	IF (MANUAL_SELECTED AND OP10B_M_PICK_PART_OK) OR OP10B_A_PICK_PART_OK THEN
		OP10B_PICK_PART_OK								:= TRUE;
		OP10B_A_ORING_INSERTION_DONE					:= TRUE;
		OP10B_Gripper_Rotate_Complete					:= TRUE;
		OP10B_Camera_Zone_Safe							:= TRUE;(*(OP10A_SRV_RH_BDYANG_CMR_FB OR OP10A_BDY2_PCK_BYPAS) AND 
															(OP10A_SRV_LH_BDYANG_CMR_FB OR OP10A_BDY1_PCK_BYPAS);*)
	ELSE
		OP10B_PICK_PART_OK								:= FALSE;
		OP10B_Gripper_Rotate_Complete					:= FALSE;
		OP10B_Camera_Zone_Safe							:= FALSE;
		OP10B_A_ORING_INSERTION_DONE					:= FALSE;		
	END_IF

	IF (MANUAL_SELECTED AND OP10B_M_PICK_PART_NOK) OR OP10B_A_PICK_PART_NOK THEN
		OP10B_PICK_PART_NOK								:= TRUE;
	ELSE
		OP10B_PICK_PART_NOK								:= FALSE;		
	END_IF

	IF (MANUAL_SELECTED AND OP10B_M_CAMERA_OK) OR OP10B_A_CAMERA_OK THEN
		OP10B_READY_TO_INSERT_ORING						:= TRUE;
		OP10B_Place_Zone_Safe							:= (OP10B_SRV_LH_BDYANG_WRK_FB OR OP10B_BDY1_PCK_BYPAS) AND 
															(OP10B_SRV_RH_BDYANG_WRK_FB OR OP10B_BDY2_PCK_BYPAS);
		OP10B_ROTATION_COMPLETE							:= TRUE;
		OP10B_O_Ring_Zone_Safe							:=  (OP10B_SRV_LH_BDYANG_FITRE_FB OR OP10B_BDY1_PCK_BYPAS) AND 
															(OP10B_SRV_RH_BDYANG_FITRE_FB OR OP10B_BDY2_PCK_BYPAS) AND 
																OP10B_CYL_RDY_TO_PLC;

		IF OP10B_ROBO_CNTRL.BDY_MVE_PLC_POS THEN
		OP10B_A_PLACE_IN_CONVEYOR						:= TRUE;			
		END_IF
		
		IF OP10B_Camera_Trigger THEN
		OP10B_CAMERA_OK									:= TRUE;	
		END_IF											
															
	ELSE                                            	
		OP10B_CAMERA_OK									:= FALSE;
		OP10B_READY_TO_INSERT_ORING						:= FALSE;
		OP10B_O_Ring_Zone_Safe							:= FALSE;
		OP10B_Place_Zone_Safe							:= FALSE;
		OP10B_A_PLACE_IN_CONVEYOR						:= FALSE;
		OP10B_ROTATION_COMPLETE							:= FALSE;		
	END_IF

	IF (MANUAL_SELECTED AND OP10B_M_CAMERA_NOK) OR OP10B_A_CAMERA_NOK AND OP10B_Camera_Trigger THEN
		OP10B_CAMERA_NOK								:= TRUE;
	ELSE
		OP10B_CAMERA_NOK								:= FALSE;		
	END_IF	 

 	IF (MANUAL_SELECTED AND OP10B_M_ORING_INSERTION_DONE) OR OP10B_A_ORING_INSERTION_DONE THEN
		OP10B_ORING_INSERTION_DONE						:= TRUE;
	ELSE
		OP10B_ORING_INSERTION_DONE						:= FALSE;		
	END_IF 
   
  	IF (MANUAL_SELECTED AND OP10B_M_PLACE_IN_CONVEYOR) OR OP10B_A_PLACE_IN_CONVEYOR THEN
		OP10B_PLACE_IN_CONVEYOR							:= TRUE;
	ELSE
		OP10B_PLACE_IN_CONVEYOR							:= FALSE;		
	END_IF

	OP10B_GRIPPER_OPEN									:= (OP10B_A_SRV_LH_GRPHME_FB OR OP10B_BDY1_PCK_BYPAS )AND (OP10B_A_SRV_RH_GRPHME_FB OR OP10B_BDY2_PCK_BYPAS) AND NOT OP10B_ROBO_Gripper_Close;
	OP10B_GRIPPER_CLOSE									:= (OP10B_A_SRV_LH_GRPWRK_FB OR  OP10B_BDY1_PCK_BYPAS)AND (OP10B_A_SRV_RH_GRPWRK_FB OR OP10B_BDY2_PCK_BYPAS) AND OP10B_ROBO_Gripper_Close;

	OP10B_Reject_Zone_Safe								:= 1;//NOT OP10A_Rbt_In_Reject_Zone;
	
//############################		OP10B STATION ENABLE CONDITION		##########################

	OP10B_STN_MOVER					:= MOVER_POSITION[OP10B_XTS_POS_NO];

	IF AUTO_WITH_XTS THEN
	IF 	OP10B_STN_MOVER>0 THEN
	IF NOT END_OF_CYCLE THEN		
	OP10B_STN_ENABLE				:= MOVER_POS_RECHED[OP10B_STN_MOVER] AND ((MOVER_CMP_STATUS[OP10B_STN_MOVER][1]=0)OR 
										(MOVER_CMP_STATUS[OP10B_STN_MOVER][2]=0))AND STATION_ENABLE_CONTROL AND NOT 
											(I10B_BDY1_PRSN_MOVER_I1001_5 OR I10B_BDY2_PRSN_MOVER_I1001_6);
  	
  
ELSE
	MOVER_CMP_STATUS[OP10B_STN_MOVER][1]					:=5;
	MOVER_CMP_STATUS[OP10B_STN_MOVER][2]					:=5;
	STATION_DONE[OP10B_STN_MOVER][OP10B_XTS_POS_NO]			:= TRUE;	
	END_IF
	ELSE	
	OP10B_STN_ENABLE				:= FALSE;
	END_IF
	END_IF

END_PROGRAM

// ---- POUs/Programs/OP10A_Bowl/Bowl_Control.TcPOU
PROGRAM Bowl_Control
VAR
	OP10A_Bowl: ModbusRtuMasterV2_KL6x22B;
	Write_Reg: UINT;
	Read: UINT;
	W_Trig	: BOOL;
	Read_Reg : UINT;
	R_Trig	: BOOL;
	Rsad:BOOL;
	Trigger: BOOL;
	R_Edge	: R_TRIG;
	reg: WORD;
	writereg: WORD;
END_VAR

//R_Edge(CLK:=W_Trig);

OP10A_Bowl.WriteSingleRegister(
	UnitID:= 1, 
	Quantity:=1 , 
	MBAddr:= writereg, 
	cbLength:= SIZEOF(Write_Reg), 
	pMemoryAddr:= ADR(Write_Reg), 
	AuxQuantity:= , 
	AuxMBAddr:= , 
	AuxcbLength:= , 
	pAuxMemoryAddr:= , 
	Execute:=W_Trig,//R_Edge.Q , 
	Timeout:= , 
	BUSY=> , 
	Error=> , 
	ErrorId=> , 
	cbRead=> );


OP10A_Bowl.ReadInputRegs(
	UnitID:= 1, 
	Quantity:=1 , 
	MBAddr:= reg, 
	cbLength:= SIZEOF(Read), 
	pMemoryAddr:= ADR(Read), 
	AuxQuantity:= , 
	AuxMBAddr:= , 
	AuxcbLength:= , 
	pAuxMemoryAddr:= , 
	Execute:=Rsad,//R_Edge.Q , 
	Timeout:= , 
	BUSY=> , 
	Error=> , 
	ErrorId=> , 
	cbRead=> );
		
	
OP10A_Bowl.ReadInputRegs(
	UnitID:= 1, 
	Quantity:=1 , 
	MBAddr:= 16#01, 
	cbLength:= SIZEOF(Read_Reg), 
	pMemoryAddr:= ADR(Read_Reg), 
	AuxQuantity:= , 
	AuxMBAddr:= , 
	AuxcbLength:= , 
	pAuxMemoryAddr:= , 
	Execute:= R_Trig, 
	Timeout:= , 
	BUSY=> , 
	Error=> , 
	ErrorId=> , 
	cbRead=> );

END_PROGRAM

// ---- POUs/Programs/OP10/OP10A_Camera_FB.TcPOU
PROGRAM OP10A_Camera_FB
VAR
	OP10A_LH_Camera 			        : FB_Cognex_ProfiNET_1;
	
	OP10A_LH_Acquisition_Status AT %I*    :Acquisition_Status;
	OP10A_LH_Inspection_Status  AT %I*    :Inspection_Status;	
	OP10A_LH_Acquisition_ID     AT %I*    :UINT;
	OP10A_LH_Inspection_ID   	 AT %I*  :UINT;
	OP10A_LH_Error_code      	 AT %I*  :UINT;
	OP10A_LH_Current_Job_ID  	 AT %I*  :UINT;
	OP10A_LH_Result_code     	 AT %I*  :UINT;
	OP10A_LH_Cam_Result      	 AT %I*  :ARRAY[0..63] OF BYTE;	
	OP10A_LH_Acquisition_Control AT %Q*  : Acquisition_Control;
	OP10A_LH_Inspection_Control  AT %Q*  : Inspection_Control;
	OP10A_LH_Command_word		AT %Q*  : UINT;
	OP10A_LH_Union                       : UNION_64Byte;

	OP10A_RH_Camera 			          : FB_Cognex_ProfiNET_1;

	
	OP10A_RH_Acquisition_Status AT %I*    :Acquisition_Status;
	OP10A_RH_Inspection_Status  AT %I*    :Inspection_Status;	
	OP10A_RH_Acquisition_ID     AT %I*    :UINT;
	OP10A_RH_Inspection_ID   	 AT %I*  :UINT;
	OP10A_RH_Error_code      	 AT %I*  :UINT;
	OP10A_RH_Current_Job_ID  	 AT %I*  :UINT;
	OP10A_RH_Result_code     	 AT %I*  :UINT;
	OP10A_RH_Cam_Result      	 AT %I*  :ARRAY[0..63] OF BYTE;	
	OP10A_RH_Acquisition_Control AT %Q*  : Acquisition_Control;
	OP10A_RH_Inspection_Control  AT %Q*  : Inspection_Control;
	OP10A_RH_Command_word		AT %Q*  : UINT;
	OP10A_RH_Union                       : UNION_64Byte;
	
	OP10_A_Empty_Camera_1	      : FB_Cognex_ProfiNET_1;
	
	
	OP10A_Empty_Cam_1_Acquisition_Status   AT %I*  :Acquisition_Status;
	OP10A_Empty_Cam_1_Inspection_Status    AT %I*  :Inspection_Status;	
	OP10A_Empty_Cam_1_Acquisition_ID       AT %I*  :UINT;
	OP10A_Empty_Cam_1_Inspection_ID   	 AT %I*  :UINT;
	OP10A_Empty_Cam_1_Error_code      	 AT %I*  :UINT;
	OP10A_Empty_Cam_1_Current_Job_ID  	 AT %I*  :UINT;
	OP10A_Empty_Cam_1_Result_code     	 AT %I*  :UINT;
	OP10A_Empty_Cam_1_Result      	 AT %I*  :ARRAY[0..63] OF BYTE;
	
	OP10A_Empty_Cam_1_Acquisition_Control AT %Q*  : Acquisition_Control;
	OP10A_Empty_Cam_1_Inspection_Control  AT %Q*  : Inspection_Control;
	OP10A_Empty_Cam_1_Command_word		AT %Q*  : UINT;
	Error_status_Cam_1						      : STRING;
	OP10A_Empty_Cam_1_Target_Job_ID				  : UINT;
	OP10A_Empty_Cam_1_Loaded_Job_ID		    	  : UINT;
	OP10A_Empty_Cam_1_Union                       : UNION_64Byte;
	OP10A_Empty_Cam_1_Job_Change_Complete		  : BOOL;
	OP10A_Empty_Cam_1_Job_Change_Error   		  : BOOL;
	OP10A_Empty_Cam_1_Picture_Taken      		  : BOOL;	
	
END_VAR

OP10A_LH_Camera (
	tTimeout:= , 
	sJob_Name:= , 
	camera_ready=> OP10A_LH_Camera_Ready,
	Camera_online=> OP10A_LH_Camera_Online,
	stCognex_record_status:=OP10A_LH_Acquisition_Status, 
	Acquisition_ID:=OP10A_LH_Acquisition_ID , 
	stCognex_Inspection_status:=OP10A_LH_Inspection_Status, 
	Error_Code:=OP10A_LH_Error_code , 
	wcommand_control_in:= OP10A_LH_Current_Job_ID, 
	aResults_64_Bytes:= OP10A_LH_Cam_Result, 
	number_of_inspections:=OP10A_LH_Inspection_ID , 
	iresult_code:= OP10A_LH_Result_code, 
	bTarget_job_ID:=OP10A_LH_Target_Job_ID , 
	Error_Status_message=> OP10A_LH_Error_status, 
	bError=> OP10A_LH_Camera_Error, 
	stCognex_record_control=>OP10A_LH_Acquisition_Control , 
	stCognex_inspection_control=>OP10A_LH_Inspection_Control , 
	wCommandControl_out=>OP10A_LH_Command_word , 
	aUser_data_64_Byte=> OP10A_LH_Union.aArrayOfByte, 
	bJob_loading_completed=>OP10A_LH_Job_Change_Complete , 
	bJob_load_failed=>OP10A_LH_Job_Change_Error , 
	bInspection_Result_IO=>  , 
	bInspection_Result_NIO=> , 
	bTXTSM_Error_Job_Change=> OP10A_LH_Job_Change_Error, 
	bPictureTakenComplete=> OP10A_LH_Picture_Taken, 
	Loaded_Job_ID=>OP10A_LH_Loaded_Job_ID	 , 
	bClear_Error:= HMI_Reset, 
	bJob_change_start:= OP10A_LH_Camera_Job_Change_start, 
	TXTSM_camera_not_online=>OP10A_LH_Camera_Error	 , 
	bTrigger_start:= OP10A_LH_Camera_Trigger );
	
OP10A_RH_Camera (
	tTimeout:= , 
	sJob_Name:= , 
	camera_ready=> OP10A_RH_Camera_Ready,
	Camera_online=> OP10A_RH_Camera_Online,
	stCognex_record_status:=OP10A_RH_Acquisition_Status, 
	Acquisition_ID:=OP10A_RH_Acquisition_ID , 
	stCognex_Inspection_status:=OP10A_RH_Inspection_Status, 
	Error_Code:=OP10A_RH_Error_code , 
	wcommand_control_in:= OP10A_RH_Current_Job_ID, 
	aResults_64_Bytes:= OP10A_RH_Cam_Result, 
	number_of_inspections:=OP10A_RH_Inspection_ID , 
	iresult_code:= OP10A_RH_Result_code, 
	bTarget_job_ID:=OP10A_RH_Target_Job_ID , 
	Error_Status_message=> OP10A_RH_Error_status, 
	bError=> OP10A_RH_Camera_Error, 
	stCognex_record_control=>OP10A_RH_Acquisition_Control , 
	stCognex_inspection_control=>OP10A_RH_Inspection_Control , 
	wCommandControl_out=>OP10A_RH_Command_word , 
	aUser_data_64_Byte=> OP10A_RH_Union.aArrayOfByte, 
	bJob_loading_completed=>OP10A_RH_Job_Change_Complete , 
	bJob_load_failed=>OP10A_RH_Job_Change_Error , 
	bInspection_Result_IO=>  , 
	bInspection_Result_NIO=> , 
	bTXTSM_Error_Job_Change=> OP10A_RH_Job_Change_Error, 
	bPictureTakenComplete=> OP10A_RH_Picture_Taken, 
	Loaded_Job_ID=>OP10A_RH_Loaded_Job_ID	 , 
	bClear_Error:= HMI_Reset, 
	bJob_change_start:= OP10A_RH_Camera_Job_Change_start, 
	TXTSM_camera_not_online=>OP10A_RH_Camera_Error	 , 
	bTrigger_start:= OP10A_RH_Camera_Trigger );	
	
OP10_A_Empty_Camera_1(
	tTimeout:= , 
	sJob_Name:= , 
	camera_ready=> OP10A_Empty_Cam_1_Camera_Ready,
	Camera_online=> OP10A_Empty_Cam_1_Camera_Online,
	stCognex_record_status:=OP10A_Empty_Cam_1_Acquisition_Status, 
	Acquisition_ID:=OP10A_Empty_Cam_1_Acquisition_ID , 
	stCognex_Inspection_status:=OP10A_Empty_Cam_1_Inspection_Status, 
	Error_Code:=OP10A_Empty_Cam_1_Error_code , 
	wcommand_control_in:= OP10A_Empty_Cam_1_Current_Job_ID, 
	aResults_64_Bytes:= OP10A_Empty_Cam_1_Result, 
	number_of_inspections:=OP10A_Empty_Cam_1_Inspection_ID , 
	iresult_code:= OP10A_Empty_Cam_1_Result_code, 
	bTarget_job_ID:=OP10A_Empty_Cam_1_Target_Job_ID , 
	Error_Status_message=> Error_status_Cam_1, 
	bError=> OP10A_Empty_Cam_1_Camera_Error, 
	stCognex_record_control=>OP10A_Empty_Cam_1_Acquisition_Control , 
	stCognex_inspection_control=>OP10A_Empty_Cam_1_Inspection_Control , 
	wCommandControl_out=>OP10A_Empty_Cam_1_Command_word , 
	aUser_data_64_Byte=> OP10A_Empty_Cam_1_Union.aArrayOfByte, 
	bJob_loading_completed=>OP10A_Empty_Cam_1_Job_Change_Complete, 
	bJob_load_failed=>OP10A_Empty_Cam_1_Job_Change_Error , 
	bInspection_Result_IO=>  , 
	bInspection_Result_NIO=> , 
	bTXTSM_Error_Job_Change=> OP10A_Empty_Cam_1_Job_Change_Error, 
	bPictureTakenComplete=> OP10A_Empty_Cam_1_Picture_Taken, 
	Loaded_Job_ID=>OP10A_Empty_Cam_1_Loaded_Job_ID	 , 
	bClear_Error:= HMI_Reset, 
	bJob_change_start:= OP10A_Empty_Cam_1_Camera_Job_Change_start, 
	TXTSM_camera_not_online=>OP10A_Empty_Cam_1_Camera_Error	 , 
	bTrigger_start:= OP10A_Empty_Cam_1_Camera_Trigger );

END_PROGRAM

// ---- FB/Cognex_Camera/FB_Cognex_ProfiNET_1.TcPOU
FUNCTION_BLOCK FB_Cognex_ProfiNET_1
VAR_INPUT
	tTimeout						: TIME := T#10S;
	sJob_Name 						: STRING(63) := '';
	stCognex_record_status     		: Acquisition_status;
	Acquisition_ID					: UINT ;//number of shots
	stCognex_Inspection_status 		: Inspection_status;
	Error_Code						: UINT ;
	wcommand_control_in 			: UINT;
    aResults_64_Bytes	     		: ARRAY[0..63] OF BYTE;
    number_of_inspections			: UINT;
	iresult_code					: UINT;
	bClear_Error					: BOOL;	
	bTarget_job_ID					: UINT;
END_VAR

VAR_OUTPUT
	Error_Status_message			:STRING;
	bError							: BOOL := 0;
	stCognex_record_control 		: Acquisition_Control;
	stCognex_inspection_control 	: Inspection_control;
    wCommandControl_out 			: UINT;
    aUser_data_64_Byte 			    : ARRAY[0..63] OF BYTE;
	bJob_loading_completed 		    : BOOL := 0; //FP
	bJob_load_failed        		: BOOL := 0; //FP
	bInspection_Result_IO 			: BOOL := 0; //FP
	bInspection_Result_NIO 			: BOOL := 0; //FP
	bTXTSM_Error_Job_Change 		: BOOL;
	bPictureTakenComplete			: BOOL;
	Loaded_Job_ID					: UINT;
	camera_ready					: BOOL;
	Camera_online					: BOOL;
	TXTSM_camera_not_online 		: BOOL := 0;
END_VAR

VAR_IN_OUT
	bJob_change_start				: BOOL := 0;	
	bTrigger_start					: BOOL := 0;
END_VAR

VAR
	ttimeout_step					: TON;
	tTimeoutStepTrigger			    : TON;
	Resul_ACk_Timer					: TON;
	//JobChange
	job_Change_OK					: R_TRIG;
	job_Change_NOK					: R_TRIG;	
	iStep_Jobchange 				: INT := 0;
	bJob_change_io 					: BOOL:= 0;
	bJob_change_nio 				: BOOL:= 0;
	//Trigger
	Trig_Start						: R_TRIG;
    iStep_Trigger				    : INT := 0;
	bInspection_io 					: BOOL:= 0;
	bInspection_nio 				: BOOL:= 0;
	bHMFPInspection_Completed		: BOOL;//HM_FP_Inspection_Completed
	bHMFNInspection_Completed		: BOOL;//HM_FN_Inspection_Completed
    
    Previous_job_id                 : UINT;   //Job ID for the last job loaded.
    Previous_job_name               : STRING; // Job name of the last job loaded.
END_VAR
VAR_TEMP
	tempaUserData_64_Byte		    : UNION_64Byte;
	bT_in 							: BOOL := FALSE;
	bT_inTrigger					: BOOL := FALSE;
	FPInspection_Completed			: BOOL := FALSE;
	FNInspection_Completed			: BOOL := FALSE;
END_VAR

stCognex_inspection_control.Buffer_Results_Enable 	:= FALSE;
stCognex_inspection_control.Inspection_Results_Ack 	:= FALSE;

Resul_ACk_Timer(IN:=stCognex_inspection_control.Inspection_Results_Ack,PT:=T#100MS);
IF Resul_ACk_Timer.Q THEN
	stCognex_inspection_control.Inspection_Results_Ack:=FALSE;
END_IF

// picture taken complete
bPictureTakenComplete:=stCognex_record_status .Exposure_Complete AND (iStep_Trigger <> 0);
stCognex_record_control.Clear_Exposure_Complete:= stCognex_record_status .Exposure_Complete;

//#########################################################################
//ErrorReset###############################################################
//#########################################################################

bError := stCognex_Inspection_status .Error;
IF bError THEN
	Previous_job_id   := 0;
    Previous_job_name := '';
END_IF

IF stCognex_Inspection_status .Error AND bClear_Error THEN
	stCognex_inspection_control.Clear_Error := TRUE;
ELSE	
	stCognex_inspection_control.Clear_Error := FALSE;
END_IF;

IF NOT stCognex_Inspection_status .Error THEN
	bClear_Error:=FALSE;
END_IF

//#########################################################################
//JobChange################################################################
//#########################################################################

CASE iStep_Jobchange OF 
	0:	//Waiting for bJob_change_start
		bJob_loading_completed := FALSE;
		bJob_load_failed := FALSE;
		bJob_change_io  := FALSE;
		bJob_change_nio := FALSE;

        // Job is still the same.
        IF (TRUE
            AND bJob_change_start
            AND (iStep_Trigger = 0)
            AND (Previous_job_id = bTarget_job_ID )
            AND (Previous_job_name = sJob_Name)
           )
        THEN
			bJob_change_start := FALSE;
            
        // Neuen Job laden.
		ELSIF bJob_change_start AND (iStep_Trigger = 0)THEN
			bJob_change_start := FALSE;
			iStep_Jobchange := 1;
		END_IF;
		
	1://Set Offline
		stCognex_record_control.Set_Offline := TRUE;
		bT_in := TRUE;
		
		IF stCognex_record_status .Online = FALSE 
			AND ( stCognex_record_status .Offline_Bit0 
					OR stCognex_record_status .Offline_Bit1 
					OR stCognex_record_status .Offline_Bit2) 
			THEN
				bT_in := FALSE;
				iStep_Jobchange := 2;
		ELSIF ttimeout_step.Q THEN //Timeout 
				bT_in := FALSE;
				iStep_Jobchange := 8;
		END_IF;
		ttimeout_step(IN:= bT_in, PT:= tTimeout, Q=> , ET=> );
		
	2://Load command(Job ID)
		wCommandControl_out := bTarget_job_ID;//4000;//
		iStep_Jobchange := 3;
		
	3://Set Job name to user data
		//FOR i:=0 TO 63 DO//initalize with 0
		//	aBenutzerdaten_64_Byte[i] := 0;
		//END_FOR;
		tempaUserData_64_Byte.sString := sJob_Name;
		aUser_data_64_Byte := tempaUserData_64_Byte.aArrayOfByte;
		iStep_Jobchange := 4;

	4://Set the Execute Command BIT in the Inspection Control Module.;
		stCognex_inspection_control.Execute_Command := TRUE;
		bT_in := TRUE;
	
		IF stCognex_Inspection_status .Command_Complete AND NOT stCognex_Inspection_status .Command_Executing THEN//Wait for result
			IF stCognex_Inspection_status .Command_Failed THEN//Job load failed 
				bT_in := FALSE;
				iStep_Jobchange := 6;
			ELSE//Job load ok
				bT_in := FALSE;
			iStep_Jobchange := 5;
			END_IF;
		ELSIF ttimeout_step.Q THEN //Timeout 
			bT_in := FALSE;
			iStep_Jobchange := 8;
		END_IF;
		ttimeout_step (IN:= bT_in, PT:= tTimeout, Q=> , ET=> );
		
	5: //Job load ok
			bT_in:= TRUE;
			stCognex_inspection_control.Execute_Command := FALSE;
			bJob_change_io := TRUE;
			bJob_change_nio := FALSE;
            
            Previous_job_id   := wcommand_control_in;
            Previous_job_name := sJob_Name;
			
		IF NOT stCognex_Inspection_status .Command_Executing THEN
			bT_in:= FALSE;
			iStep_Jobchange := 7;
		ELSIF ttimeout_step.Q THEN //Timeout 
			bT_in := FALSE;
			iStep_Jobchange := 8;
		END_IF;
		ttimeout_step(IN:= bT_in, PT:= tTimeout, Q=> , ET=> );
			
	6:	//Job load failed
			bT_in:= TRUE;
			stCognex_inspection_control.Execute_Command := FALSE;
			bJob_change_io := FALSE;
			bJob_change_nio := TRUE;
            
            Previous_job_id   := 0;
            Previous_job_name := '';
			
		IF NOT stCognex_Inspection_status .Command_Executing THEN
			bT_in:= FALSE;
			iStep_Jobchange := 7;
		ELSIF ttimeout_step.Q THEN //Timeout 
			bT_in := FALSE;
			iStep_Jobchange := 8;
		END_IF;
		ttimeout_step(IN:= bT_in, PT:= tTimeout, Q=> , ET=> );
			
	7://Set online 
		bT_in := TRUE;
		stCognex_record_control.Set_Offline := FALSE;
		
		IF stCognex_record_status .Online = TRUE THEN
			iStep_Jobchange := 9;
			bT_in := FALSE;
		ELSIF ttimeout_step.Q THEN //Timeout 
			iStep_Jobchange := 8;
			bT_in := FALSE;
		END_IF;
		ttimeout_step(IN:= bT_in, PT:= tTimeout, Q=> , ET=> );
		
	8://Global Timeout
			stCognex_record_control.Set_Offline := FALSE;
			stCognex_inspection_control.Execute_Command := FALSE;
			bJob_change_io := FALSE;
			bJob_change_nio := TRUE;
			iStep_Jobchange := 9;
			
	9://Set Output signals
	 IF bTarget_job_ID=Loaded_Job_ID  THEN
		bJob_loading_completed:=1;
	 ELSE
	 	bJob_load_failed:=1;
	 END_IF

		//bJob_loading_completed := bJob_change_io;
		//bJob_load_failed := bJob_change_nio;
		iStep_Jobchange := 0;
	ELSE //CASE JobChange default
		
	iStep_Jobchange := 0;
	
END_CASE;

//output error messages Job-change

IF bJob_change_nio THEN
	bTXTSM_Error_Job_Change := TRUE;
	Previous_job_id   := 0;
    Previous_job_name := '';
ELSIF (bJob_change_io AND NOT bJob_change_nio) OR bClear_Error THEN
	bTXTSM_Error_Job_Change := FALSE;
END_IF;

	// IF bTarget_job_ID=Loaded_Job_ID  THEN
	//	bJob_loading_completed:=1;
	// ELSE
	// 	bJob_load_failed:=1;
	// END_IF
//#########################################################################
//Trigger##################################################################
//#########################################################################
//Inspection_Completed edge (Toggle)
FPInspection_Completed 		:= stCognex_Inspection_status .Inspection_Completed AND NOT bHMFPInspection_Completed ;
bHMFPInspection_Completed 	:= stCognex_Inspection_status .Inspection_Completed;

FNInspection_Completed := NOT stCognex_Inspection_status .Inspection_Completed AND bHMFNInspection_Completed ;
bHMFNInspection_Completed := 	stCognex_Inspection_status .Inspection_Completed;
//Camera waiting for result:
IF iStep_Trigger = 2
	 OR iStep_Trigger = 3
	 OR iStep_Trigger = 4 
THEN
	IF (FPInspection_Completed OR FNInspection_Completed) THEN
        IF stCognex_Inspection_status .Results_Valid THEN // stCognex_Inspection_status .Job_Pass THEN
		    bInspection_io  := TRUE;
		    bInspection_nio := FALSE;
			stCognex_inspection_control.Inspection_Results_Ack :=TRUE;
        ELSE
		    bInspection_io  := FALSE;
		    bInspection_nio := TRUE;
			stCognex_inspection_control.Inspection_Results_Ack :=TRUE;
        END_IF
	END_IF
(* PHU: von ARU
	IF (FPInspection_Completed OR FNInspection_Completed) AND stCognex_Inspektionsstatus.Job_Pass THEN
		bInspection_io := TRUE; 
	ELSIF (FPInspection_Completed OR FNInspection_Completed) AND NOT stCognex_Inspektionsstatus.Job_Pass THEN
		bInspection_nio := TRUE; 
	END_IF
*)
END_IF
CASE iStep_Trigger OF 
	0:	//Waiting for bTrigger_start
		bInspection_Result_IO := FALSE;
		bInspection_Result_NIO := FALSE;
		bInspection_io  := FALSE;
		bInspection_nio := FALSE;
		
		Trig_Start(CLK:=bTrigger_start);
		IF Trig_Start.Q AND (iStep_Jobchange = 0) AND NOT bTXTSM_Error_Job_Change THEN
			bTrigger_start := FALSE;
			iStep_Trigger := 1;
		END_IF;
	1://Enable External Trigger
		stCognex_record_control.Trigger_Enable := TRUE;
		stCognex_record_control.Trigger := FALSE;
		//stCognex_Aufnahmesteuerung.Trigger := FALSE;
		
		IF  stCognex_record_status .Trigger_Ready AND stCognex_record_status .Online AND NOT  stCognex_Inspection_status .System_Busy THEN//NOT stCognex_Inspektionsstatus.Command_Executing THEN
			iStep_Trigger := 2;
			
		END_IF;
	2://Trigger start
	
		
		stCognex_record_control.Trigger := TRUE;
		bT_inTrigger:= TRUE;
		
		IF stCognex_record_status .Trigger_Ack THEN
			bT_inTrigger := FALSE;
			iStep_Trigger := 3;
		ELSIF tTimeoutStepTrigger.Q THEN //Timeout 
			bT_inTrigger := FALSE;
			iStep_Trigger := 0;
		END_IF
		
		tTimeoutStepTrigger(IN:= bT_inTrigger, PT:= T#30S, Q=> , ET=> );		
		
	3://Trigger Reset	
		stCognex_record_control.Trigger := FALSE;
		bT_inTrigger:= TRUE;
		
		IF stCognex_record_status .Trigger_Ack = FALSE THEN
			bT_inTrigger := FALSE;
			iStep_Trigger := 4;
		ELSIF tTimeoutStepTrigger.Q THEN //Timeout 
			bT_inTrigger := FALSE;
			iStep_Trigger := 0;
		END_IF;
		
		tTimeoutStepTrigger(IN:= bT_inTrigger, PT:= T#30S, Q=> , ET=> );
		
	4://Wait for result
	
		bT_inTrigger:= TRUE;
	
		IF bInspection_io OR bInspection_nio THEN
			bT_inTrigger:= FALSE;
			iStep_Trigger := 5;
		ELSIF tTimeoutStepTrigger.Q THEN //Timeout 
			bT_inTrigger := FALSE;
			iStep_Trigger := 0;
		END_IF;
		
		tTimeoutStepTrigger(IN:= bT_inTrigger, PT:= T#30S, Q=> , ET=> );
	
	5://Set Output signals
		IF bInspection_nio = TRUE THEN
			bInspection_Result_NIO	:= TRUE; 
			bInspection_Result_IO	:= FALSE;
			iStep_Trigger := 0; 
		ELSIF bInspection_io THEN
			bInspection_Result_NIO	:= FALSE; 
			bInspection_Result_IO	:= TRUE; 
			iStep_Trigger := 0;
		END_IF;


	ELSE //CASE Trigger default
		
	iStep_Trigger := 0;

END_CASE;

camera_ready:=stCognex_record_status.Trigger_Ready;
Camera_online:=	stCognex_record_status.Online;
Loaded_Job_ID:=wcommand_control_in;

//#########################################################################
//output error messages##################################################
//#########################################################################

TXTSM_camera_not_online
 := (NOT ( stCognex_record_status .Offline_Bit0 AND stCognex_record_status .Offline_Bit1 AND NOT stCognex_record_status .Offline_Bit2) 
AND (NOT (iStep_Jobchange = 7))							
AND (NOT stCognex_record_status .Online));

IF TXTSM_camera_not_online
 THEN
   Previous_job_id   := 0;
   Previous_job_name := '';
END_IF;

IF Error_Code=0 AND NOT TXTSM_camera_not_online THEN
	Error_Status_message:= 'No Error and Camera Online';
ELSIF TXTSM_camera_not_online THEN
	Error_Status_message:='Camera_Offline';
ELSIF Error_Code= 256 THEN
	Error_Status_message:='Error_0x0100-Trigger set while disabled';
ELSIF Error_Code= 257 THEN
	Error_Status_message:='Error_0x0101-Trigger set while offline';
ELSIF Error_Code= 1024 THEN
	Error_Status_message:='Error_0x0400-Job change executing bit is always High';
ELSIF Error_Code= 1025 THEN
	Error_Status_message:='Error_0x0401-Job change requested while online';
ELSIF Error_Code= 1026 THEN
	Error_Status_message:='Error_0x0402-Requestd job is not saved';	
ELSIF Error_Code= 1040 THEN
	Error_Status_message:='Error_0x0410-Testrun disabled';
ELSIF Error_Code= 1041 THEN
	Error_Status_message:='Error_0x0411-Testrun requested while online';	
END_IF

END_FUNCTION_BLOCK

// ---- POUs/Programs/OP10/OP10B_Camera_FB.TcPOU
PROGRAM OP10B_Camera_FB
VAR
	OP10B_LH_Camera 			        : FB_Cognex_ProfiNET_1;

	
	OP10B_LH_Acquisition_Status AT %I*    :Acquisition_Status;
	OP10B_LH_Inspection_Status  AT %I*    :Inspection_Status;	
	OP10B_LH_Acquisition_ID     AT %I*    :UINT;
	OP10B_LH_Inspection_ID   	 AT %I*  :UINT;
	OP10B_LH_Error_code      	 AT %I*  :UINT;
	OP10B_LH_Current_Job_ID  	 AT %I*  :UINT;
	OP10B_LH_Result_code     	 AT %I*  :UINT;
	OP10B_LH_Cam_Result      	 AT %I*  :ARRAY[0..63] OF BYTE;	
	OP10B_LH_Acquisition_Control AT %Q*  : Acquisition_Control;
	OP10B_LH_Inspection_Control  AT %Q*  : Inspection_Control;
	OP10B_LH_Command_word		AT %Q*  : UINT;
	OP10B_LH_Union                       : UNION_64Byte;

	OP10B_RH_Camera 			          : FB_Cognex_ProfiNET_1;

	
	OP10B_RH_Acquisition_Status AT %I*    :Acquisition_Status;
	OP10B_RH_Inspection_Status  AT %I*    :Inspection_Status;	
	OP10B_RH_Acquisition_ID     AT %I*    :UINT;
	OP10B_RH_Inspection_ID   	 AT %I*  :UINT;
	OP10B_RH_Error_code      	 AT %I*  :UINT;
	OP10B_RH_Current_Job_ID  	 AT %I*  :UINT;
	OP10B_RH_Result_code     	 AT %I*  :UINT;
	OP10B_RH_Cam_Result      	 AT %I*  :ARRAY[0..63] OF BYTE;	
	OP10B_RH_Acquisition_Control AT %Q*  : Acquisition_Control;
	OP10B_RH_Inspection_Control  AT %Q*  : Inspection_Control;
	OP10B_RH_Command_word		AT %Q*  : UINT;
	OP10B_RH_Union                       : UNION_64Byte;
	
	OP10_B_Empty_Camera_2	      : FB_Cognex_ProfiNET_1;

	
	OP10B_Empty_Cam_2_Acquisition_Status   AT %I*  :Acquisition_Status;
	OP10B_Empty_Cam_2_Inspection_Status    AT %I*  :Inspection_Status;	
	OP10B_Empty_Cam_2_Acquisition_ID       AT %I*  :UINT;
	OP10B_Empty_Cam_2_Inspection_ID   	 AT %I*  :UINT;
	OP10B_Empty_Cam_2_Error_code      	 AT %I*  :UINT;
	OP10B_Empty_Cam_2_Current_Job_ID  	 AT %I*  :UINT;
	OP10B_Empty_Cam_2_Result_code     	 AT %I*  :UINT;
	OP10B_Empty_Cam_2_Result      	 AT %I*  :ARRAY[0..63] OF BYTE;
	
	OP10B_Empty_Cam_2_Acquisition_Control AT %Q*  : Acquisition_Control;
	OP10B_Empty_Cam_2_Inspection_Control  AT %Q*  : Inspection_Control;
	OP10B_Empty_Cam_2_Command_word		AT %Q*  : UINT;
	Error_status_Cam_2						      : STRING;
	OP10B_Empty_Cam_2_Target_Job_ID				  : UINT;
	OP10B_Empty_Cam_2_Loaded_Job_ID		    	  : UINT;
	OP10B_Empty_Cam_2_Union                       : UNION_64Byte;
	OP10B_Empty_Cam_2_Job_Change_Complete		  : BOOL;
	OP10B_Empty_Cam_2_Job_Change_Error   		  : BOOL;
	OP10B_Empty_Cam_2_Picture_Taken      		  : BOOL;	
END_VAR

OP10B_LH_Camera (
	tTimeout:= , 
	sJob_Name:= , 
	camera_ready=> OP10B_LH_Camera_Ready,
	Camera_online=> OP10B_LH_Camera_Online,
	stCognex_record_status:=OP10B_LH_Acquisition_Status, 
	Acquisition_ID:=OP10B_LH_Acquisition_ID , 
	stCognex_Inspection_status:=OP10B_LH_Inspection_Status, 
	Error_Code:=OP10B_LH_Error_code , 
	wcommand_control_in:= OP10B_LH_Current_Job_ID, 
	aResults_64_Bytes:= OP10B_LH_Cam_Result, 
	number_of_inspections:=OP10B_LH_Inspection_ID , 
	iresult_code:= OP10B_LH_Result_code, 
	bTarget_job_ID:=OP10B_LH_Target_Job_ID , 
	Error_Status_message=> OP10B_LH_Error_status, 
	bError=> OP10B_LH_Camera_Error, 
	stCognex_record_control=>OP10B_LH_Acquisition_Control , 
	stCognex_inspection_control=>OP10B_LH_Inspection_Control , 
	wCommandControl_out=>OP10B_LH_Command_word , 
	aUser_data_64_Byte=> OP10B_LH_Union.aArrayOfByte, 
	bJob_loading_completed=>OP10B_LH_Job_Change_Complete , 
	bJob_load_failed=>OP10B_LH_Job_Change_Error , 
	bInspection_Result_IO=>  , 
	bInspection_Result_NIO=> , 
	bTXTSM_Error_Job_Change=> OP10B_LH_Job_Change_Error, 
	bPictureTakenComplete=> OP10B_LH_Picture_Taken, 
	Loaded_Job_ID=>OP10B_LH_Loaded_Job_ID	 , 
	bClear_Error:= HMI_Reset, 
	bJob_change_start:= OP10B_LH_Camera_Job_Change_start, 
	TXTSM_camera_not_online=>OP10B_LH_Camera_Error	 , 
	bTrigger_start:= OP10B_LH_Camera_Trigger );
	
OP10B_RH_Camera (
	tTimeout:= , 
	sJob_Name:= , 
	camera_ready=> OP10B_RH_Camera_Ready,
	Camera_online=> OP10B_RH_Camera_Online,
	stCognex_record_status:=OP10B_RH_Acquisition_Status, 
	Acquisition_ID:=OP10B_RH_Acquisition_ID , 
	stCognex_Inspection_status:=OP10B_RH_Inspection_Status, 
	Error_Code:=OP10B_RH_Error_code , 
	wcommand_control_in:= OP10B_RH_Current_Job_ID, 
	aResults_64_Bytes:= OP10B_RH_Cam_Result, 
	number_of_inspections:=OP10B_RH_Inspection_ID , 
	iresult_code:= OP10B_RH_Result_code, 
	bTarget_job_ID:=OP10B_RH_Target_Job_ID , 
	Error_Status_message=> OP10B_RH_Error_status, 
	bError=> OP10B_RH_Camera_Error, 
	stCognex_record_control=>OP10B_RH_Acquisition_Control , 
	stCognex_inspection_control=>OP10B_RH_Inspection_Control , 
	wCommandControl_out=>OP10B_RH_Command_word , 
	aUser_data_64_Byte=> OP10B_RH_Union.aArrayOfByte, 
	bJob_loading_completed=>OP10B_RH_Job_Change_Complete , 
	bJob_load_failed=>OP10B_RH_Job_Change_Error , 
	bInspection_Result_IO=>  , 
	bInspection_Result_NIO=> , 
	bTXTSM_Error_Job_Change=> OP10B_RH_Job_Change_Error, 
	bPictureTakenComplete=> OP10B_RH_Picture_Taken, 
	Loaded_Job_ID=>OP10B_RH_Loaded_Job_ID	 , 
	bClear_Error:= HMI_Reset, 
	bJob_change_start:= OP10B_RH_Camera_Job_Change_start, 
	TXTSM_camera_not_online=>OP10B_RH_Camera_Error	 , 
	bTrigger_start:= OP10B_RH_Camera_Trigger );	

OP10_B_Empty_Camera_2(
	tTimeout:= , 
	sJob_Name:= , 
	camera_ready=> OP10B_Empty_Cam_2_Camera_Ready,
	Camera_online=> OP10B_Empty_Cam_2_Camera_Online,
	stCognex_record_status:=OP10B_Empty_Cam_2_Acquisition_Status, 
	Acquisition_ID:=OP10B_Empty_Cam_2_Acquisition_ID , 
	stCognex_Inspection_status:=OP10B_Empty_Cam_2_Inspection_Status, 
	Error_Code:=OP10B_Empty_Cam_2_Error_code , 
	wcommand_control_in:= OP10B_Empty_Cam_2_Current_Job_ID, 
	aResults_64_Bytes:= OP10B_Empty_Cam_2_Result, 
	number_of_inspections:=OP10B_Empty_Cam_2_Inspection_ID , 
	iresult_code:= OP10B_Empty_Cam_2_Result_code, 
	bTarget_job_ID:=OP10B_Empty_Cam_2_Target_Job_ID , 
	Error_Status_message=> Error_status_Cam_2, 
	bError=> OP10B_Empty_Cam_2_Camera_Error, 
	stCognex_record_control=>OP10B_Empty_Cam_2_Acquisition_Control , 
	stCognex_inspection_control=>OP10B_Empty_Cam_2_Inspection_Control , 
	wCommandControl_out=>OP10B_Empty_Cam_2_Command_word , 
	aUser_data_64_Byte=> OP10B_Empty_Cam_2_Union.aArrayOfByte, 
	bJob_loading_completed=>OP10B_Empty_Cam_2_Job_Change_Complete, 
	bJob_load_failed=>OP10B_Empty_Cam_2_Job_Change_Error , 
	bInspection_Result_IO=>  , 
	bInspection_Result_NIO=> , 
	bTXTSM_Error_Job_Change=> OP10B_Empty_Cam_2_Job_Change_Error, 
	bPictureTakenComplete=> OP10B_Empty_Cam_2_Picture_Taken, 
	Loaded_Job_ID=>OP10B_Empty_Cam_2_Loaded_Job_ID	 , 
	bClear_Error:= HMI_Reset, 
	bJob_change_start:= OP10B_Empty_Cam_2_Camera_Job_Change_start, 
	TXTSM_camera_not_online=>OP10B_Empty_Cam_2_Camera_Error	 , 
	bTrigger_start:= OP10B_Empty_Cam_2_Camera_Trigger );

END_PROGRAM

// ---- POUs/Programs/OP10/OP10A_OP10B_DRUM_FEEDER.TcPOU
PROGRAM OP10A_OP10B_DRUM_FEEDER
VAR
	OP10A_DRUM_FB					: Servo_Conveyor_FB;
	OP10B_DRUM_FB					: Servo_Conveyor_FB;
		
	OP10A_CONVEYOR_ON				: BOOL;
	OP10B_CONVEYOR_ON				: BOOL;
	OP10A_DRUM_CNVY_CNTINUS_RUN		: BOOL;	
	OP10A_VELOCITY_MODE				: BOOL;
	OP10A_CAMERA_TRIG				: BOOL;
	OP10A_COVY_OVER_FLOW			: BOOL;
	OP10A_Onecycle					: BOOL;
	OP10_A_Camera_Done : BOOL;
	Conveyor_Track_Delay: TON;
	Conveyor_Track_OFF_Delay: TON;

	OP10B_Conveyor_Track_Delay: TON;
	OP10B_Conveyor_Track_OFF_Delay: TON;
	
	OP10A_Conveyor_Control: BOOL;
	OP10B_DRUM_CNVY_CNTINUS_RUN: BOOL;
	OP10_B_Camera_Done: BOOL;
	OP10B_Onecycle: BOOL;
	OP10B_Conveyor_Control: BOOL;

	cge: BOOL;
END_VAR

VAR PERSISTENT
	OP10A_OVR_FLW_TIMER				: TIME;
	OP10A_CONVY_FRWD_SPD			: REAL;
	OP10A_CONVY_REV_SPD				: REAL;
	OP10A_FWD_POS_DISTANCE			: REAL;
	OP10A_REV_POS_DISTANCE			: REAL;
	OP10A_CONV_FRWD_TIME			: INT;	
	OP10A_CONV_REV_TIME				: INT;	

	OP10B_FWD_POS_DISTANCE          : REAL;
	OP10B_REV_POS_DISTANCE			: REAL;

END_VAR


//O10A_DRUM_MTR_FWD_Q708_4				:=I10A_DRUM_OFF_ON_I714_2;
//O10A_DRUM_FEED_AIRPURGE_ON_Q1052_1		:=O10A_DRUM_MTR_FWD_Q708_4;

IF MANUAL_SELECTED AND OP10A_MANUAL_SELECTED THEN               
	IF I10A_DRUM_CONV_REV_I714_3 THEN
		OP10A_SRV_O_CNVY_STUS.targetVelocity:=OP10A_CONVY_REV_SPD;
		OP10A_SRV_O_CNVY_STUS.moveVelocity:=I10A_DRUM_CONV_REV_I714_3;
 	ELSIF I10A_DRUM_CONV_FWD_I714_4 THEN
		OP10A_SRV_O_CNVY_STUS.targetVelocity:= OP10A_CONVY_FRWD_SPD;
		OP10A_SRV_O_CNVY_STUS.moveVelocity:=I10A_DRUM_CONV_FWD_I714_4;	
	ELSE 	
		OP10A_SRV_O_CNVY_STUS.moveVelocity:=0;   	
	END_IF  	
END_IF  

IF MANUAL_SELECTED AND OP10B_MANUAL_SELECTED THEN               
	IF I10B_DRUM_CONV_REV_I302_3 THEN
		OP10B_SRV_O_CNVY_STUS.targetVelocity:= OP10A_CONVY_REV_SPD;
		OP10B_SRV_O_CNVY_STUS.moveVelocity:=I10B_DRUM_CONV_REV_I302_3;
 	ELSIF I10B_DRUM_CONV_FWD_I302_4 THEN
		OP10B_SRV_O_CNVY_STUS.targetVelocity:=OP10A_CONVY_FRWD_SPD;
		OP10B_SRV_O_CNVY_STUS.moveVelocity:=I10B_DRUM_CONV_FWD_I302_4;	
	ELSE 	
		OP10B_SRV_O_CNVY_STUS.moveVelocity:=0;   	
	END_IF  	
END_IF  

OP10A_DRUM_FB(
	Conveyor_Prgrm_Start:= OP10A_AUTO_RUNNING , 
	Conveyor_Prgrm_Reset:= , 
	Conveyor_Continuous_Run:= OP10A_DRUM_CNVY_CNTINUS_RUN , 
	Conveyor_Bypass:= ,
	Camera_Trigger_OK := OP10A_Camera_Done, 
	Fwd_Time_IP:= OP10A_CONV_FRWD_TIME, 
	Rev_Time_IP:= OP10A_CONV_REV_TIME, 
	Conveyor_FWD_Speed:= OP10A_CONVY_FRWD_SPD, 
	Conveyor_REV_Speed:= OP10A_CONVY_REV_SPD, 
	Conveyor_FWD_Position:= OP10A_FWD_POS_DISTANCE, 
	Conveyor_REV_Position:= OP10A_REV_POS_DISTANCE, 
	Velocity_mode:= OP10A_VELOCITY_MODE, 
	LH_Work_Sensor:= OP10A_LH_REJ.Sensor2, 
	LH_Home_Sensor:= OP10A_LH_REJ.Sensor1, 
	RH_Work_Sensor:= OP10A_RH_REJ.Sensor2,  
	RH_Home_Sensor:= OP10A_RH_REJ.Sensor1,
	LH_Camera_OK:= OP10A_LH_CMR_OK , 
	LH_Camera_NOK:= OP10A_LH_CMR_NOK, 
	RH_Camera_OK:= OP10A_RH_CMR_OK , 
	RH_Camera_NOK:= OP10A_RH_CMR_NOK, 
	Track_Overflow := Conveyor_Track_OFF_Delay.Q,
	Track_Sensor_FB := Conveyor_Track_Delay.Q,
	Camera_Trigger_Ack=> OP10A_Camera_Trigger_Ack,
	Camera_trigger:= OP10A_Camera_Trigger, 
	LH_Work_Coil=> OP10A_A_LH_REJ_WRK, 
	LH_Home_Coil=> OP10A_A_LH_REJ_HOME, 
	RH_Work_Coil=> OP10A_A_RH_REJ_WRK, 
	RH_Home_Coil=> OP10A_A_RH_REJ_HOME, 
	Drum_ON=> O10A_DRUM_MTR_FWD_Q708_4,
	Step_Num => Conv_Step_no_10A,
	Ready_to_Pick=> OP10A_ORNG_RDY_PCK, 
	One_Cycle:= OP10A_Onecycle, 
	Pick_Done:= OP10A_ORNG_PCK_DN,  
	Conveyor_Servo_Control_Structure:= OP10A_SRV_O_CNVY_CNT);
	


Conveyor_Track_Delay(IN:= NOT I10A_DRUM_LH_CONV_OVR_FLW_I1010_0 AND NOT I10A_DRUM_RH_CONV_OVR_FLW_I1010_1,PT:=T#4S);	
Conveyor_Track_OFF_Delay(IN:=I10A_DRUM_LH_CONV_OVR_FLW_I1010_0 AND I10A_DRUM_RH_CONV_OVR_FLW_I1010_1,PT:=T#1S);   

IF OP10A_Conveyor_Control THEN
	IF Conveyor_Track_OFF_Delay.Q THEN
		O10A_DRUM_MTR_FWD_Q708_4:=0;
	END_IF
	//IF Conveyor_Track_Delay.Q THEN
	//	O10A_DRUM_MTR_FWD_Q708_4:=1;
	//END_IF
	O10A_DRUM_FEED_AIRPURGE_ON_Q1052_1:=1;
	O10A_DRUM_RUN_IND_Q709_0:=O10A_DRUM_MTR_FWD_Q708_4;
ELSE
	O10A_DRUM_MTR_FWD_Q708_4:=I10A_DRUM_OFF_ON_I714_2;
    O10A_DRUM_RUN_IND_Q709_0:=I10A_DRUM_OFF_ON_I714_2;
    O10A_DRUM_FEED_AIRPURGE_ON_Q1052_1 :=I10A_DRUM_OFF_ON_I714_2;
END_IF
	
	
OP10B_DRUM_FB(
	Conveyor_Prgrm_Start:= OP10B_AUTO_RUNNING , 
	Conveyor_Prgrm_Reset:= , 
	Conveyor_Continuous_Run:= OP10B_DRUM_CNVY_CNTINUS_RUN , 
	Conveyor_Bypass:= ,
	Camera_Trigger_OK := OP10B_Camera_Done, 
	Fwd_Time_IP:= OP10A_CONV_FRWD_TIME, 
	Rev_Time_IP:= OP10A_CONV_REV_TIME, 
	Conveyor_FWD_Speed:= OP10A_CONVY_FRWD_SPD, 
	Conveyor_REV_Speed:= OP10A_CONVY_REV_SPD, 
	Conveyor_FWD_Position:= OP10A_FWD_POS_DISTANCE, 
	Conveyor_REV_Position:= OP10A_REV_POS_DISTANCE, 
	Velocity_mode:= OP10A_VELOCITY_MODE, 
	LH_Work_Sensor:= OP10B_LH_REJ.Sensor2, 
	LH_Home_Sensor:= OP10B_LH_REJ.Sensor1, 
	RH_Work_Sensor:= OP10B_RH_REJ.Sensor2,  
	RH_Home_Sensor:= OP10B_RH_REJ.Sensor1,
	LH_Camera_OK:= OP10A_LH_CMR_OK , 
	LH_Camera_NOK:= OP10A_LH_CMR_NOK, 
	RH_Camera_OK:= OP10A_RH_CMR_OK , 
	RH_Camera_NOK:= OP10A_RH_CMR_NOK, 
	Track_Overflow := OP10B_Conveyor_Track_OFF_Delay.Q,
	Track_Sensor_FB := OP10B_Conveyor_Track_Delay.Q,
	Camera_Trigger_Ack=> OP10B_Camera_Trigger_Ack,
	Camera_trigger:= OP10B_Camera_Trigger,
	Step_Num => Conv_Step_no_10B, 
	LH_Work_Coil=> OP10B_A_LH_REJ_WRK, 
	LH_Home_Coil=> OP10B_A_LH_REJ_HOME, 
	RH_Work_Coil=> OP10B_A_RH_REJ_WRK, 
	RH_Home_Coil=> OP10B_A_RH_REJ_HOME, 
	Drum_ON=> O10B_DRUM_MTR_FWD_Q302_0,
	Ready_to_Pick=> OP10B_ORNG_RDY_PCK,
	One_Cycle:= OP10B_Onecycle, 
	Pick_Done:=OP10B_ORNG_PCK_DN,  
	Conveyor_Servo_Control_Structure:= OP10B_SRV_O_CNVY_CNT);	
	
OP10B_Conveyor_Track_Delay(IN:= NOT I10B_DRUM_LH_CONV_OVR_FLW_I1030_0 AND NOT I10B_DRUM_RH_CONV_OVR_FLW_I1030_1,PT:=T#4S);	
OP10B_Conveyor_Track_OFF_Delay(IN:=I10B_DRUM_LH_CONV_OVR_FLW_I1030_0 AND I10B_DRUM_RH_CONV_OVR_FLW_I1030_1,PT:=T#1S);   

IF OP10B_Conveyor_Control THEN
	IF OP10B_Conveyor_Track_OFF_Delay.Q THEN
		O10B_DRUM_MTR_FWD_Q302_0:=0;
	END_IF
	//IF Conveyor_Track_Delay.Q THEN
	//	O10A_DRUM_MTR_FWD_Q708_4:=1;
	//END_IF
	O10B_DRUM_FEED_AIRPURGE_ON_Q1062_0:=1;
	O10B_DRUM_RUN_IND_Q302_4:=O10B_DRUM_MTR_FWD_Q302_0;
ELSE
	O10B_DRUM_MTR_FWD_Q302_0:=I10B_DRUM_OFF_ON_I302_2;
    O10B_DRUM_RUN_IND_Q302_4:=I10B_DRUM_OFF_ON_I302_2;
    O10B_DRUM_FEED_AIRPURGE_ON_Q1062_0 :=I10B_DRUM_OFF_ON_I302_2;
END_IF

END_PROGRAM

// ---- FB/Servo_Conveyor_FB.TcPOU
FUNCTION_BLOCK Servo_Conveyor_FB
VAR_INPUT
	Conveyor_Prgrm_Start			: BOOL;
	Conveyor_Prgrm_Reset			: BOOL;
	Conveyor_Continuous_Run			: BOOL;	
	Camera_Trigger_OK				: BOOL;	
	Conveyor_Bypass					: BOOL;
	Fwd_Time_IP						: INT;
	Rev_Time_IP						: INT;
	Conveyor_FWD_Speed				: REAL;
	Conveyor_REV_Speed				: REAL;
	Conveyor_FWD_Position			: REAL;
	Conveyor_REV_Position			: REAL;	
	Velocity_mode					: BOOL;
	LH_Work_Sensor					: BOOL;
	LH_Home_Sensor					: BOOL;
	RH_Work_Sensor					: BOOL;
	RH_Home_Sensor					: BOOL;	
	LH_Camera_OK					: BOOL;
	LH_Camera_NOK					: BOOL;	
	RH_Camera_OK					: BOOL;
	RH_Camera_NOK					: BOOL;
	Track_Overflow					: BOOL;
	Track_Sensor_FB					: BOOL;
END_VAR
VAR_OUTPUT
	Camera_Trigger_ACK				: BOOL;	
	LH_Work_Coil					: BOOL;
	LH_Home_Coil					: BOOL;
	RH_Work_Coil					: BOOL;
	RH_Home_Coil					: BOOL;	
	Ready_to_Pick					: BOOL;
	Drum_ON							: BOOL;
	Step_Num						: INT;
END_VAR
VAR_IN_OUT
	Camera_trigger						: BOOL;
	One_Cycle							: BOOL;
	Pick_Done						    : BOOL;
	Conveyor_Servo_Control_Structure	:  Servo_Control;
END_VAR
VAR
	Conveyor_Speed  : REAL;
	Cyl_Delay 		: TON;
	Cyl_Temp 		: BOOL;
	temp_3			: BOOL;
	cam_ok 			: BOOL;
	con_step_no 	: INT;	
	t1				: ton;
	t2				: ton;
	t3				: ton;
	t4				: ton;	
	count_nok   	: INT;
	forward			: BOOL;
	reverse			: BOOL;
	fwd_time		: INT;
	rev_time		: INT;
	temp            : BOOL;
	VeloCity_Frwd   : REAL := 200;
	Track_Count		: TON;
	Temp_1 : R_TRIG;
	Temp_Cont : BOOL;
	
END_VAR

IF NOT Conveyor_Prgrm_Start OR Conveyor_Servo_Control_Structure.Axis_Error THEN
	con_step_no:=10;
	Ready_to_Pick:=FALSE;
	Conveyor_Servo_Control_Structure.VELmove_Start:=FALSE;
END_IF

IF Conveyor_Bypass THEN
	con_step_no:=10;
	Ready_to_Pick:=1;
	IF Pick_Done THEN
		Pick_Done:=0;
		Ready_to_Pick:=0;
	END_IF
END_IF

IF forward THEN
	Conveyor_Speed:=Conveyor_FWD_Speed;
END_IF
IF reverse THEN
	Conveyor_Speed:=Conveyor_REV_Speed;
END_IF

CASE con_step_no OF
		10: IF Conveyor_Prgrm_Start THEN
				con_step_no:=15;
			END_IF
			
		15: LH_Home_Coil:=1;
			RH_Home_Coil:=1;	
			IF LH_Home_Sensor AND RH_Home_Sensor THEN
				LH_Home_Coil:=0;
				RH_Home_Coil:=0;
				con_step_no:= 20;
			END_IF
		
        20:	Ready_to_Pick :=FALSE;
			Pick_Done:= FALSE;
			Conveyor_Servo_Control_Structure.Velocity:= VeloCity_Frwd;		
			Conveyor_Servo_Control_Structure.VELmove_Start:=FALSE;
			IF NOT Conveyor_Servo_Control_Structure.VELmove_Start THEN
				con_step_no:= 25;
			END_IF	
			
		25:	Drum_ON:=1;
			Conveyor_Servo_Control_Structure.VELmove_Start:=TRUE;	
			IF Track_Overflow THEN
				Conveyor_Servo_Control_Structure.VELmove_Start:=FALSE;
				Drum_ON	   :=FALSE;
				con_step_no:= 80;
			END_IF
	
		  
		70: IF NOT Conveyor_Servo_Control_Structure.VELmove_Start THEN
			  Camera_trigger :=TRUE;
			  con_step_no	 := 75;
			END_IF	
					
		75:	IF Camera_Trigger_OK AND NOT Conveyor_Servo_Control_Structure.VELmove_Start AND Conveyor_Servo_Control_Structure.Axis_ready THEN
				IF LH_Camera_OK AND RH_Camera_OK THEN
				 con_step_no:= 100;
				 fwd_time:=Fwd_Time_IP;
				 count_nok:=0;	
				ELSIF (LH_Camera_NOK)  AND RH_Camera_OK AND count_nok<5 THEN
				 count_nok := count_nok +1;
				 con_step_no:= 76;	
				ELSIF (RH_Camera_NOK) AND LH_Camera_OK AND count_nok<5 THEN
				 count_nok := count_nok +1;
				 con_step_no:= 78;	 
				ELSIF RH_Camera_NOK AND LH_Camera_NOK AND count_nok<5 THEN
				 count_nok := count_nok +1;
				 con_step_no:= 101;	  
				ELSIF count_nok>=5 THEN
	             fwd_time:=3000;
				 con_step_no:= 80; 
				END_IF
			END_IF	
			
		76:	IF  NOT Conveyor_Servo_Control_Structure.VELmove_Start THEN
				IF LH_Home_Sensor THEN
					LH_Work_Coil:=TRUE;
					Cyl_Temp:=1;
				END_IF	
				IF Cyl_Delay.Q THEN
					con_step_no:= 77;
				END_IF				
			END_IF	
			
		77: 	IF  LH_Work_Sensor THEN
					LH_Work_Coil:=0;
					LH_Home_Coil:=1;
				END_IF	
				IF LH_Home_Sensor AND NOT LH_Work_Coil AND count_nok<5 THEN
					LH_Home_Coil:=0;
					fwd_time:=Fwd_Time_IP;
				    con_step_no:= 80;
				END_IF
                IF  LH_Home_Sensor AND NOT LH_Work_Coil AND count_nok>=5 THEN
					LH_Home_Coil:=0;
					fwd_time:=3000;
					count_nok:=0;
				    con_step_no:= 80;	
				END_IF

		78:	IF NOT Conveyor_Servo_Control_Structure.VELmove_Start THEN	
				IF RH_Home_Sensor THEN
					RH_Work_Coil:=TRUE;
					Cyl_Temp:=1;
				END_IF	
				IF Cyl_Delay.Q THEN
					con_step_no:= 79;
				END_IF				
			END_IF		
			
		79: 	IF RH_Work_Sensor THEN
					RH_Work_Coil:=0;
					RH_Home_Coil:=1;				
				END_IF
				IF RH_Home_Sensor AND NOT RH_Work_Coil AND count_nok<5 THEN
					RH_Home_Coil:=0;					
					fwd_time:=Fwd_Time_IP;
				    con_step_no:= 80;
				END_IF
				IF RH_Home_Sensor AND NOT RH_Work_Coil AND count_nok>=5 THEN
					fwd_time:=3000;
					count_nok:=0;
					RH_Home_Coil:=0;
				    con_step_no:= 80;	
				END_IF
			
		80: 	IF Velocity_mode THEN
					IF fwd_time=3000 THEN
			       		count_nok:=0;	
					END_IF
                	Conveyor_Servo_Control_Structure.Velocity:= Conveyor_Speed;				
					forward:=TRUE;
					Conveyor_Servo_Control_Structure.VELmove_Start:=TRUE;	
					IF t2.Q THEN
    					forward:=FALSE;
						Conveyor_Servo_Control_Structure.VELmove_Start:=FALSE;
						Camera_Trigger_ACK:=1;
						con_step_no:= 90;
					END_IF
				ELSE
					Conveyor_Servo_Control_Structure.Velocity:=Conveyor_FWD_Speed;
					Conveyor_Servo_Control_Structure.Position:=Conveyor_FWD_Position;
					Conveyor_Servo_Control_Structure.RELmove_Start:=1;
					con_step_no:= 85;
				END_IF	
				
		85 : 	IF NOT Conveyor_Servo_Control_Structure.RELmove_Start THEN 
					con_step_no:= 90;
				END_IF	
		
		90: IF Velocity_mode THEN
				Conveyor_Servo_Control_Structure.Velocity:= Conveyor_Speed;
				reverse:=TRUE;
				Conveyor_Servo_Control_Structure.VELmove_Start:=TRUE;
				IF t3.Q THEN
 					reverse:=FALSE;
					Conveyor_Servo_Control_Structure.VELmove_Start:=FALSE;
					con_step_no:= 70;
				END_IF
			ELSE
				Conveyor_Servo_Control_Structure.Velocity:=ABS(Conveyor_REV_Speed);
				Conveyor_Servo_Control_Structure.Position:=(-Conveyor_REV_Position);
				Conveyor_Servo_Control_Structure.RELmove_Start:=1;
				con_step_no:= 92;
			END_IF
			
		91:  IF NOT Camera_Trigger_OK THEN
				Camera_Trigger_ACK:=0;
				con_step_no:= 70;
			 END_IF		
			
		92 : 	IF NOT Conveyor_Servo_Control_Structure.RELmove_Start THEN 
					Camera_Trigger_ACK:=0;
					con_step_no:= 70;
				END_IF
				
		100: IF NOT Conveyor_Servo_Control_Structure.VELmove_Start THEN
				 Camera_Trigger_ACK:=1;
				 Ready_to_Pick:=TRUE;
			 END_IF	
			 IF Pick_Done OR Conveyor_Continuous_Run THEN
				 Ready_to_Pick :=FALSE;
				 Pick_Done:= FALSE;
				 con_step_no:= 80;
			 END_IF	

		101: IF LH_Home_Sensor AND RH_Home_Sensor THEN
					LH_Work_Coil:=TRUE;
					RH_Work_Coil:=TRUE;
					Cyl_Temp:=1;
				END_IF	
				IF Cyl_Delay.Q THEN
					con_step_no:= 102;
				END_IF	

		102: IF RH_Work_Sensor AND LH_Work_Sensor THEN
					RH_Work_Coil:=0;
					LH_Work_Coil:=0;
					RH_Home_Coil:=1;
					LH_Home_Coil:=1;				
				END_IF
				IF RH_Home_Sensor AND LH_Home_Sensor AND NOT RH_Work_Coil AND NOT LH_Work_Coil AND count_nok<5 THEN
					RH_Home_Coil:=0;	
					LH_Home_Coil:=0;				
					fwd_time:=Fwd_Time_IP;
				    con_step_no:= 80;
				END_IF	
				IF RH_Home_Sensor AND LH_Home_Sensor AND NOT RH_Work_Coil AND NOT LH_Work_Coil AND count_nok>=5 THEN
					RH_Home_Coil:=0;	
					LH_Home_Coil:=0;				
					fwd_time:=3000;
				    con_step_no:= 80;
				END_IF		
END_CASE

Track_Count(IN:=Track_Sensor_FB,PT:=T#5S);
IF Track_Sensor_FB AND ( con_step_no=100 ) AND NOT Conveyor_Servo_Control_Structure.VELmove_Start THEN
	con_step_no:= 20;
END_IF

Step_Num:=con_step_no;
	
Temp_1(CLK:=Track_Count.Q );
//t1(IN:=Camera_trigger ,PT:=T#500MS);

//IF Camera_trigger AND con_step_no=70  THEN
//	Camera_Trigger_OK:=FALSE;
//END_IF

//IF t1.Q THEN
//	Camera_Trigger_OK:=1;
//	Camera_trigger :=FALSE;
//END_IF

temp:=1;
rev_time:=Rev_Time_IP;

t2(IN:=forward ,PT:=INT_TO_TIME(fwd_time));
t3(IN:=reverse ,PT:=INT_TO_TIME(rev_time));
//t4(IN:=Camera_trigger,PT:=T#500MS);

Cyl_Delay(IN:=Cyl_Temp,PT:=T#600MS);
IF Cyl_Delay.Q THEN
	Cyl_Temp:=0;
END_IF

IF One_Cycle THEN
	con_step_no := 80;
	One_Cycle	:=0;
END_IF

END_FUNCTION_BLOCK

// ---- POUs/Programs/OP10/OP10B_Conveyor_Prog.TcPOU
PROGRAM OP10B_Conveyor_Prog
VAR
	Conv_Cam_Step : INT;
	Temp_Counter_LH : UINT;
	Temp_Counter_RH : UINT;
	Toggle_Pos : R_TRIG;
	Toggle_Neg : F_TRIG;
END_VAR

CASE Conv_Cam_Step OF
	10: 	OP10B_LH_Camera_OK :=0;
            OP10B_LH_Camera_NOK:=0;
	        OP10B_RH_Camera_OK :=0;
	        OP10B_RH_Camera_NOK:=0;			
			OP10B_Camera_Done	:=0;
			//OP10B_LH_Clr_OK 		:=0;
		   // OP10B_RH_Clr_OK 		:=0;		
			//OP10B_LH_Size_OK		:=0;
		    //OP10B_RH_Size_OK		:=0;	
			Conv_Cam_Step		:=11;	
	
	11: IF (OP10B_Camera_Trigger AND (NOT OP10B_Camera_Done)) OR OP10B_Miss_Trigger THEN
			OP10B_LH_Camera_Trigger:=1;
			OP10B_RH_Camera_Trigger:=1;
			Conv_Cam_Step		  :=15;	
		END_IF

	15:	IF Toggle_Pos.Q OR Toggle_Neg.Q THEN// (NOT OP10B_LH_Camera_Trigger) AND (NOT OP10B_RH_Camera_Trigger) THEN //(Temp_Counter_LH<OP10B_Camera_FB.OP10B_LH_Acquisition_ID AND Temp_Counter_RH<OP10B_Camera_FB.OP10B_RH_Acquisition_ID )THEN
			OP10B_LH_Camera_Trigger:=0;
			OP10B_RH_Camera_Trigger:=0;
			OP10B_Camera_Trigger :=0;
			OP10B_Miss_Trigger	:=0;
			Conv_Cam_Step:=25;
		END_IF  
	   
	25: IF OP10B_Camera_FB.OP10B_LH_Cam_Result[0]=1 AND OP10B_Camera_FB.OP10B_RH_Cam_Result[0]=1 THEN
			OP10B_LH_Camera_OK:=1;
			OP10B_RH_Camera_OK:=1;
			Conv_Cam_Step    :=50;
		ELSIF (OP10B_Camera_FB.OP10B_LH_Cam_Result[1]=1 OR OP10B_Camera_FB.OP10B_RH_Cam_Result[1]=1) THEN //AND ( OP10B_Camera_FB.OP10B_LH_Cam_Result[2]=1 AND OP10B_Camera_FB.OP10B_RH_Cam_Result[2]=1) THEN			
			IF OP10B_Camera_FB.OP10B_LH_Cam_Result[0]=1 THEN
				OP10B_LH_Camera_OK:=1;
			END_IF
			IF OP10B_Camera_FB.OP10B_RH_Cam_Result[0]=1 THEN
				OP10B_RH_Camera_OK:=1;
			END_IF
			Conv_Cam_Step:=30;
		END_IF	
			
   30: 	IF OP10B_Camera_FB.OP10B_LH_Cam_Result[1]=1 THEN
	   		OP10B_LH_Camera_NOK:=1;
  	    END_IF
		IF OP10B_Camera_FB.OP10B_RH_Cam_Result[1]=1 THEN
	   		OP10B_RH_Camera_NOK:=1;
  	    END_IF
		Conv_Cam_Step:=50;
		
   50:  OP10B_Camera_Done:=1;
   		Temp_Counter_LH:=OP10B_Camera_FB.OP10B_LH_Acquisition_ID;
		Temp_Counter_RH:=OP10B_Camera_FB.OP10B_RH_Acquisition_ID;
		IF Conv_Step_no_10B>75 THEN
			Conv_Cam_Step   :=10;
			OP10B_Camera_Done:=0;
		END_IF
   	    
END_CASE

Toggle_Pos(CLK:=OP10B_Camera_FB.OP10B_LH_Inspection_Status.Inspection_Completed);
Toggle_Neg(CLK:=OP10B_Camera_FB.OP10B_LH_Inspection_Status.Inspection_Completed);

END_PROGRAM

// ---- POUs/Programs/OP10/OP10A_Conveyor_Prog.TcPOU
PROGRAM OP10A_Conveyor_Prog
VAR
	Conv_Cam_Step : INT;
	Temp_Counter_LH : UINT;
	Temp_Counter_RH : UINT;
	Toggle_Pos : R_TRIG;
	Toggle_Neg : F_TRIG;

END_VAR

CASE Conv_Cam_Step OF
	10: 	OP10A_LH_Camera_OK :=0;
            OP10A_LH_Camera_NOK:=0;
	        OP10A_RH_Camera_OK :=0;
	        OP10A_RH_Camera_NOK:=0;			
			OP10A_Camera_Done	:=0;
			//OP10A_LH_Clr_OK 		:=0;
		   // OP10A_RH_Clr_OK 		:=0;		
			//OP10A_LH_Size_OK		:=0;
		    //OP10A_RH_Size_OK		:=0;	
			Conv_Cam_Step		:=11;	
	
	11: IF (OP10A_Camera_Trigger AND (NOT OP10A_Camera_Done)) OR OP10A_Miss_Trigger THEN
			OP10A_LH_Camera_Trigger:=1;
			OP10A_RH_Camera_Trigger:=1;
			Conv_Cam_Step		  :=15;	
		END_IF

	15:	IF Toggle_Pos.Q OR Toggle_Neg.Q THEN// (NOT OP10A_LH_Camera_Trigger) AND (NOT OP10A_RH_Camera_Trigger) THEN //(Temp_Counter_LH<OP10A_Camera_FB.OP10A_LH_Acquisition_ID AND Temp_Counter_RH<OP10A_Camera_FB.OP10A_RH_Acquisition_ID )THEN
			OP10A_LH_Camera_Trigger:=0;
			OP10A_RH_Camera_Trigger:=0;
			OP10A_Camera_Trigger :=0;
			OP10A_Miss_Trigger	:=0;
			Conv_Cam_Step:=25;
		END_IF  
	   
	25: IF OP10A_Camera_FB.OP10A_LH_Cam_Result[0]=1 AND OP10A_Camera_FB.OP10A_RH_Cam_Result[0]=1 THEN
			OP10A_LH_Camera_OK:=1;
			OP10A_RH_Camera_OK:=1;
			Conv_Cam_Step    :=50;
		ELSIF (OP10A_Camera_FB.OP10A_LH_Cam_Result[1]=1 OR OP10A_Camera_FB.OP10A_RH_Cam_Result[1]=1) THEN //AND ( OP10A_Camera_FB.OP10A_LH_Cam_Result[2]=1 AND OP10A_Camera_FB.OP10A_RH_Cam_Result[2]=1) THEN			
			IF OP10A_Camera_FB.OP10A_LH_Cam_Result[0]=1 THEN
				OP10A_LH_Camera_OK:=1;
			END_IF
			IF OP10A_Camera_FB.OP10A_RH_Cam_Result[0]=1 THEN
				OP10A_RH_Camera_OK:=1;
			END_IF
			Conv_Cam_Step:=30;
		END_IF	
			
   30: 	IF OP10A_Camera_FB.OP10A_LH_Cam_Result[1]=1 THEN
	   		OP10A_LH_Camera_NOK:=1;
  	    END_IF
		IF OP10A_Camera_FB.OP10A_RH_Cam_Result[1]=1 THEN
	   		OP10A_RH_Camera_NOK:=1;
  	    END_IF
		Conv_Cam_Step:=50;
		
   50:  OP10A_Camera_Done:=1;
   		Temp_Counter_LH:=OP10A_Camera_FB.OP10A_LH_Acquisition_ID;
		Temp_Counter_RH:=OP10A_Camera_FB.OP10A_RH_Acquisition_ID;
		IF Conv_Step_no_10A>75 THEN
			Conv_Cam_Step   :=10;
			OP10A_Camera_Done:=0;
		END_IF
   	    
END_CASE

Toggle_Pos(CLK:=OP10A_Camera_FB.OP10A_LH_Inspection_Status.Inspection_Completed);
Toggle_Neg(CLK:=OP10A_Camera_FB.OP10A_LH_Inspection_Status.Inspection_Completed);

END_PROGRAM

// ---- POUs/Programs/OP10/Body_Singulation_Seq.TcPOU
PROGRAM Body_Singulation_Seq
VAR

	AFT_GRP_HME_10A			: TON;
	AFT_SRV_WRK_10A			: TON;
	AFT_GRP_WRK_10A			: TON;
	Part_Presnce_Delay_10A  : TON;
	AFT_GRP_HME_10B			: TON;
	AFT_SRV_WRK_10B			: TON;
	AFT_GRP_WRK_10B			: TON;
	Part_Presnce_Delay_10B  : TON;

	
	Toggle_Pos_LH_Empty : R_TRIG;
	Toggle_Neg_LH_Empty : F_TRIG;
	Toggle_Pos_RH_Empty : R_TRIG;
	Toggle_Neg_RH_Empty : F_TRIG;	
	OP10B_Empty_Cam_Completed : BOOL;
	OP10A_Empty_Cam_Completed : BOOL;	
	Singulation_Seq_Start_manual     : BOOL;
	
	Bowl_A_ON_Timer		: TON;
	Bowl_A_OFF_Timer	: TON;
	Bowl_B_ON_Timer		: TON;
	Bowl_B_OFF_Timer	: TON;	
	
	
END_VAR

VAR PERSISTENT
	Str_variant 			: BOOL;
	OP10A_Camera_Bypass     : BOOL;
	OP10A_angle_Bypass      : BOOL;
	OP10A_singulation_Bypass: BOOL;

	OP10B_Camera_Bypass     : BOOL;
	OP10B_angle_Bypass      : BOOL;
	OP10B_singulation_Bypass: BOOL;	
	
	AFT_GRP_HME_TIME			: TIME ;
	AFT_SRV_WRK_TIME			: TIME ;
	AFT_GRP_WRK_TIME			: TIME ;
	AFT_Part_Prsnce_TIME		: TIME;	
	
	OP10A_Bowl_On_time			: TIME;
	OP10A_Bowl_OFF_time			: TIME;
	
	OP10B_Bowl_On_time			: TIME;
	OP10B_Bowl_OFF_time			: TIME;
END_VAR

IF OP10A_ERR OR OP10B_ERR THEN
	OP10A_Sing_Seq:=10;	
    OP10B_Sing_Seq:=10;
		//OP10_A_SRV_FST_BDYPCK_WRK		:= FALSE;//((NOT CHECK) OR 
		//OP10_A_SRV_SCND_BDYPCK_WRK		:= FALSE;
		OP10_A_FRT_BDY_SING_HME			:= FALSE; 
		OP10_A_SEC_BDY_SING_HME			:= FALSE; 
		OP10_A_FRT_BDY_SING_WRK			:= FALSE;
		OP10_A_SEC_BDY_SING_WRK			:= FALSE;
		OP10_LH_CMP_RDY_PCK				:= FALSE;
		OP10_RH_CMP_RDY_PCK				:= FALSE;
		OP10_A_SRV_FST_BDYPCK_WRK		:= FALSE;
		OP10_A_SRV_FST_BDYPCK_HME       := FALSE;
		OP10_A_SRV_SCND_BDYPCK_WRK      := FALSE;
		OP10_A_SRV_SCND_BDYPCK_HME      := FALSE;
		//OP10_A_SRV_SCND_BDYPCK_HME		:= FALSE;	
		//OP10_A_SRV_FST_BDYPCK_HME		:= FALSE;	
END_IF

//NOT Singulation_Seq_Start_manual AND

Toggle_Pos_RH_Empty(CLK:=OP10A_Camera_FB.OP10A_Empty_Cam_1_Inspection_Status.Inspection_Completed);
Toggle_Neg_RH_Empty(CLK:=OP10A_Camera_FB.OP10A_Empty_Cam_1_Inspection_Status.Inspection_Completed);
IF Toggle_Pos_RH_Empty.Q OR Toggle_Pos_RH_Empty.Q THEN
	OP10A_Empty_Cam_Completed:=1;	
END_IF

Toggle_Pos_LH_Empty(CLK:=OP10B_Camera_FB.OP10B_Empty_Cam_2_Inspection_Status.Inspection_Completed);
Toggle_Neg_LH_Empty(CLK:=OP10B_Camera_FB.OP10B_Empty_Cam_2_Inspection_Status.Inspection_Completed);
IF Toggle_Pos_LH_Empty.Q OR Toggle_Pos_LH_Empty.Q THEN
	OP10B_Empty_Cam_Completed:=1;	
END_IF

AFT_GRP_HME_10A(IN:=OP10_BDY_SING_FRT.Sensor1,PT:=AFT_GRP_HME_TIME);
AFT_SRV_WRK_10A(IN:=OP10_SRV_FRST_PCKBDY_WRK_FB,PT:=AFT_SRV_WRK_TIME);
AFT_GRP_WRK_10A(IN:=OP10_BDY_SING_FRT.Sensor2,PT:=AFT_GRP_WRK_TIME);
Part_Presnce_Delay_10A(IN:= I10_RH_LNR_TRK_BDY_PRSN_I1000_6,PT:=AFT_Part_Prsnce_TIME );

AFT_GRP_HME_10B(IN:=OP10_BDY_SING_SEC.Sensor1,PT:=AFT_GRP_HME_TIME);
AFT_SRV_WRK_10B(IN:=OP10_SRV_SCND_PCKBDY_WRK_FB,PT:=AFT_SRV_WRK_TIME);
AFT_GRP_WRK_10B(IN:=OP10_BDY_SING_SEC.Sensor2,PT:=AFT_GRP_WRK_TIME);
Part_Presnce_Delay_10B(IN:= I10_LH_LNR_TRK_BDY_PRSN_I1000_5,PT:=AFT_Part_Prsnce_TIME );

CASE OP10A_Sing_Seq OF
	10: IF ( (OP10A_AUTO_RUNNING OR OP10A_STEP_RUNNING) OR (OP10B_AUTO_RUNNING OR OP10B_STEP_RUNNING)) AND NOT OP10A_singulation_Bypass THEN
		   OP10A_Sing_Seq:=15;
		ELSIF OP10A_singulation_Bypass THEN
    	   OP10A_Sing_Seq:=180;
		END_IF
		
	15:	IF OP10_COMP_PICKED_1 THEN
		    OP10A_Sing_Seq:=120;
		ELSE
			OP10A_Sing_Seq:=20;	
		END_IF
	
	20: OP10_A_FRT_BDY_SING_HME	:=1;
		OP10_A_FRT_BDY_SING_WRK :=0;
		OP10_A_SRV_FST_BDYPCK_HME := TRUE;	   
		IF OP10_BDY_SING_FRT.Sensor1 AND OP10_SRV_FRST_PCKBDY_HME_FB THEN
			OP10_A_FRT_BDY_SING_HME	:=0;
			IF AFT_GRP_HME_10A.Q THEN
				OP10A_Sing_Seq:=40;
			END_IF	
		END_IF		
		
	40: IF Part_Presnce_Delay_10A. Q AND NOT OP10B_Rbt_In_Pick_Zone AND NOT OP10A_Rbt_In_Pick_Zone THEN 
			OP10A_Sing_Seq:=60;
		END_IF
	
	60: OP10_A_SRV_FST_BDYPCK_WRK		:= TRUE;
		IF AFT_SRV_WRK_10A.Q THEN
			OP10A_Sing_Seq:=80;
		END_IF
		
   80: OP10_A_FRT_BDY_SING_WRK  :=1;
   	   OP10_A_FRT_BDY_SING_HME	:=0;
   	   IF AFT_GRP_WRK_10A.Q THEN
		   OP10_A_FRT_BDY_SING_WRK :=0;
		   OP10A_Sing_Seq:=100;
	   END_IF
 
  100: OP10_A_SRV_FST_BDYPCK_HME := TRUE;
	   IF OP10_SRV_FRST_PCKBDY_HME_FB THEN
		   OP10A_Sing_Seq:=120;
	   END_IF
	   
 120: 	OP10A_Empty_Cam_Completed:=0;  
		OP10A_Body_OK	         :=0;	
		OP10A_Body_NOK			 :=0;
		OP10A_Body_Window_0Deg	 :=0;
		OP10A_Body_Window_90Deg	 :=0;
	 	OP10A_Sing_Seq:=130; 
	  
 130: OP10A_Empty_Cam_1_Camera_Trigger:=Pulse_Block.Q10Hz;
	  IF OP10A_Empty_Cam_Completed AND NOT OP10A_Camera_Bypass THEN
	 	OP10A_Sing_Seq:=140;
	  ELSIF OP10A_Empty_Cam_Completed AND OP10A_Camera_Bypass THEN
		OP10A_Body_OK			:=1;
		OP10A_Body_Window_0Deg  :=1;
		OP10A_Sing_Seq:=180;	
 	  END_IF
		  
 140: IF OP10A_Camera_FB.OP10A_Empty_Cam_1_Result[1]=1 THEN
	 	OP10A_Body_OK:=1;
		OP10A_Sing_Seq:=160;
	  ELSIF OP10A_Camera_FB.OP10A_Empty_Cam_1_Result[1]=0 THEN	
		OP10A_Body_NOK    :=1;
		OP10_COMP_PICKED_1:=0;
		OP10A_Sing_Seq    :=10;
 	  END_IF
			     	   
 160: IF OP10A_Body_OK AND OP10A_Camera_FB.OP10A_Empty_Cam_1_Result[0]=1 AND NOT OP10A_angle_Bypass AND Str_variant THEN
	 	OP10A_Body_Window_0Deg := 1;
		OP10A_Sing_Seq		   :=180;
	  ELSIF OP10A_Body_OK AND OP10A_Camera_FB.OP10A_Empty_Cam_1_Result[0]=2 AND NOT OP10A_angle_Bypass AND Str_variant THEN
	 	OP10A_Body_Window_90Deg := 1;
		OP10A_Sing_Seq		    :=180; 	
	  ELSIF OP10A_angle_Bypass OR (NOT Str_variant) THEN
		OP10A_Body_Window_0Deg := 1;
		OP10A_Sing_Seq		   :=180;
	  END_IF	
	
  180:   OP10_RH_CMP_RDY_PCK:=1;    
	     OP10_COMP_PICKED_1 :=1; 
	     OP10A_Sing_Seq	 :=200;
	  
  200:  IF ((OP10A_A_SRV_RH_GRPWRK_FB OR OP10A_BDY2_PCK_BYPAS) AND (OP10A_A_SRV_LH_GRPWRK_FB OR OP10A_BDY1_PCK_BYPAS) AND OP10A_Rbt_In_Pick_Zone) 
			OR ((OP10B_A_SRV_LH_GRPWRK_FB OR OP10B_BDY1_PCK_BYPAS) AND (OP10B_A_SRV_RH_GRPWRK_FB OR OP10B_BDY2_PCK_BYPAS) AND OP10B_Rbt_In_Pick_Zone) THEN
	  	   OP10_A_FRT_BDY_SING_HME	:=1;
		   OP10_A_FRT_BDY_SING_WRK :=0;
		   OP10_RH_CMP_RDY_PCK :=0; 
		   IF OP10_BDY_SING_FRT.Sensor1 THEN
				OP10_A_FRT_BDY_SING_HME	:=0;
				IF AFT_GRP_HME_10A.Q THEN
		 			 OP10A_Sing_Seq :=220;
				END_IF	
	   	   END_IF
 		 END_IF		

  220:  IF (NOT OP10B_Rbt_In_Pick_Zone AND NOT OP10A_Rbt_In_Pick_Zone) THEN  
		  OP10_COMP_PICKED_1  :=0;
		  OP10A_Sing_Seq      :=10;
	    END_IF	 
	  
END_CASE

CASE OP10B_Sing_Seq OF
	10: IF((OP10A_AUTO_RUNNING OR OP10A_STEP_RUNNING) OR (OP10B_AUTO_RUNNING OR OP10B_STEP_RUNNING)) AND NOT OP10B_singulation_Bypass THEN
		   OP10B_Sing_Seq:=15;
		ELSIF OP10B_singulation_Bypass THEN
    	   OP10B_Sing_Seq:=180;
		END_IF
	
	15: IF OP10_COMP_PICKED_2 THEN
		    OP10B_Sing_Seq:=120;
		ELSE
			OP10B_Sing_Seq:=20;
		END_IF
		
	20: OP10_A_SEC_BDY_SING_HME	:=1;
		OP10_A_SEC_BDY_SING_WRK :=0;
		OP10_A_SRV_SCND_BDYPCK_HME := TRUE;
		IF OP10_BDY_SING_SEC.Sensor1 AND OP10_SRV_SCND_PCKBDY_HME_FB THEN
			OP10_A_SEC_BDY_SING_HME	:=0;
			IF AFT_GRP_HME_10B.Q THEN
				OP10B_Sing_Seq:=40;
			END_IF	
		END_IF		
		
	40: IF Part_Presnce_Delay_10B. Q AND NOT OP10B_Rbt_In_Pick_Zone AND NOT OP10A_Rbt_In_Pick_Zone THEN 
			OP10B_Sing_Seq:=60;
		END_IF
	
	60: OP10_A_SRV_SCND_BDYPCK_WRK	:= TRUE;
		IF AFT_SRV_WRK_10B.Q THEN
			OP10B_Sing_Seq:=80;
		END_IF
		
   80: OP10_A_SEC_BDY_SING_WRK  :=1;
   	   OP10_A_SEC_BDY_SING_HME	:=0;
   	   IF AFT_GRP_WRK_10B.Q THEN
		  OP10_A_SEC_BDY_SING_WRK :=0;
		  OP10B_Sing_Seq:=100;
	   END_IF
 
  100: OP10_A_SRV_SCND_BDYPCK_HME := TRUE;
	   IF OP10_SRV_SCND_PCKBDY_HME_FB THEN
		   OP10B_Sing_Seq:=120;
	   END_IF
	   
 120: 	OP10B_Empty_Cam_Completed:=0;  
		OP10B_Body_OK	         :=0;	
		OP10B_Body_NOK			 :=0;
		OP10B_Body_Window_0Deg	 :=0;
		OP10B_Body_Window_90Deg	 :=0;
	 	OP10B_Sing_Seq			 :=130; 
	  
 130: OP10B_Empty_Cam_2_Camera_Trigger:=Pulse_Block.Q10Hz;
	  IF OP10B_Empty_Cam_Completed AND NOT OP10B_Camera_Bypass THEN
	 	OP10B_Sing_Seq			:=140;
	  ELSIF OP10B_Empty_Cam_Completed AND OP10B_Camera_Bypass THEN
		OP10B_Body_OK			:=1;
		OP10B_Body_Window_0Deg  :=1;
		OP10B_Sing_Seq	        :=180;	
 	  END_IF
		  
 140: IF OP10B_Camera_FB.OP10B_Empty_Cam_2_Result[1]=1 THEN
	 	OP10B_Body_OK  :=1;
		OP10B_Sing_Seq :=160;
	  ELSIF OP10B_Camera_FB.OP10B_Empty_Cam_2_Result[1]=0 THEN	
		OP10B_Body_NOK     :=1;
		OP10_COMP_PICKED_2 :=0;
		OP10B_Sing_Seq     :=10;
 	  END_IF
			     	   
 160: IF OP10B_Body_OK AND OP10B_Camera_FB.OP10B_Empty_Cam_2_Result[0]=1 AND NOT OP10B_angle_Bypass AND Str_variant THEN
	 	OP10B_Body_Window_0Deg  := 1;
		OP10B_Sing_Seq		    :=180;
	  ELSIF OP10B_Body_OK AND OP10B_Camera_FB.OP10B_Empty_Cam_2_Result[0]=2 AND NOT OP10B_angle_Bypass AND Str_variant THEN
	 	OP10B_Body_Window_90Deg := 1;
		OP10B_Sing_Seq		    :=180; 	
	  ELSIF OP10B_angle_Bypass OR (NOT Str_variant) THEN
		OP10B_Body_Window_0Deg  := 1;
		OP10B_Sing_Seq		    :=180;
	  END_IF	
	
   180: OP10_LH_CMP_RDY_PCK:=1;  
 	  	OP10_COMP_PICKED_2:=1;
	    OP10B_Sing_Seq    :=200;
	  
   200: IF ((OP10A_A_SRV_RH_GRPWRK_FB OR OP10A_BDY2_PCK_BYPAS) AND (OP10A_A_SRV_LH_GRPWRK_FB OR OP10A_BDY1_PCK_BYPAS) AND OP10A_Rbt_In_Pick_Zone) 
			OR ((OP10B_A_SRV_LH_GRPWRK_FB OR OP10B_BDY1_PCK_BYPAS) AND (OP10B_A_SRV_RH_GRPWRK_FB OR OP10B_BDY2_PCK_BYPAS) AND OP10B_Rbt_In_Pick_Zone) THEN	   		OP10_A_SEC_BDY_SING_HME :=1;
   	   		OP10_A_SEC_BDY_SING_WRK	:=0;
			OP10_A_SEC_BDY_SING_HME :=1;
		 	OP10_LH_CMP_RDY_PCK:=0;		
			IF AFT_GRP_HME_10B.Q THEN
		 		OP10_A_SEC_BDY_SING_HME :=0;
		  		OP10B_Sing_Seq:=220;
	        END_IF
   		END_IF
	  
   220:	IF (NOT OP10B_Rbt_In_Pick_Zone AND NOT OP10A_Rbt_In_Pick_Zone) THEN

		  OP10_COMP_PICKED_2:=0;
		  OP10B_Sing_Seq    :=10;
	  	END_IF 
		
END_CASE

O10A_BDY_LNR1_AIR_PURGE_Q101_3:=I10A_BDY_BWL_RUN_I101_3;
O10A_BDY_LNR2_AIR_PURGE_Q101_4:=I10A_BDY_BWL_RUN_I101_3;
O10B_BDY_LNR1_AIR_PURGE_Q201_3:=I10B_BDY_BWL_RUN_I201_3;
O10B_BDY_LNR2_AIR_PURGE_Q201_4:=I10B_BDY_BWL_RUN_I201_3;

O10A_HPR_MTR_FWD_Q100_0			:=I10A_HPR_OFF_ON_I100_4;
O10A_HPR_TWR_LMP_GREEN_Q100_6	:=I10A_HPR_OFF_ON_I100_4;
//O10A_BDY_BOWL_ON_Q101_0			:=I10A_BDY_BOWL_OFF_ON_I100_5;
O10A_BDY_LNR_FEED1_ON_Q101_1	:=I10A_BDY_LNR1_OFF_ON_I100_6 OR I10A_BDY_LNR2_OFF_ON_I100_7;
O10A_BDY_LNR_FEED2_ON_Q101_2    :=I10A_BDY_LNR1_OFF_ON_I100_6 OR I10A_BDY_LNR2_OFF_ON_I100_7;

O10B_HPR_MTR_FWD_Q200_0		   := I10B_HPR_OFF_ON_I200_4;
O10B_HPR_TWR_LMP_GREEN_Q200_6  := I10B_HPR_OFF_ON_I200_4;
//O10B_BDY_BOWL_ON_Q201_0        := I10B_BDY_BOWL_OFF_ON_I200_5;
O10B_BDY_LNR_FEED1_ON_Q201_1   := I10B_BDY_LNR1_OFF_ON_I200_6 OR I10B_BDY_LNR2_OFF_ON_I200_7;
O10B_BDY_LNR_FEED2_ON_Q201_2   := I10B_BDY_LNR1_OFF_ON_I200_6 OR I10B_BDY_LNR2_OFF_ON_I200_7;

Bowl_A_ON_Timer(IN:= NOT I10A_BDY_LNR_FEED1_OVRFLW_I101_6,PT:=OP10A_Bowl_On_time);
Bowl_A_OFF_Timer(IN:= I10A_BDY_LNR_FEED1_OVRFLW_I101_6,PT:=OP10A_Bowl_OFF_time);

Bowl_B_ON_Timer(IN:= NOT I10B_BDY_LNR_FEED1_OVRFLW_I201_6,PT:=OP10B_Bowl_On_time);
Bowl_B_OFF_Timer(IN:=I10B_BDY_LNR_FEED1_OVRFLW_I201_6,PT:=OP10B_Bowl_OFF_time);

//Bowl_A_ON_Timer(IN:= NOT I10A_BDY_LNR_FEED2_OVRFLW_I101_7,PT:=T#2S);
//Bowl_A_OFF_Timer(IN:= I10A_BDY_LNR_FEED1_OVRFLW_I101_6,PT:=T#2S);
//
//Bowl_B_ON_Timer(IN:= NOT I10B_BDY_LNR_FEED2_OVRFLW_I201_7,PT:=T#2S);
//Bowl_B_OFF_Timer(IN:=I10B_BDY_LNR_FEED1_OVRFLW_I201_6,PT:=T#2S);

IF I10A_BDY_BOWL_OFF_ON_I100_5 THEN
	IF 	Bowl_A_OFF_Timer.Q THEN
		O10A_BDY_BOWL_ON_Q101_0:=1;
	END_IF
	IF Bowl_A_ON_Timer.Q THEN
		O10A_BDY_BOWL_ON_Q101_0:=0;
	END_IF
ELSE
	O10A_BDY_BOWL_ON_Q101_0:=1;
END_IF

IF I10B_BDY_BOWL_OFF_ON_I200_5 THEN
	IF 	Bowl_B_OFF_Timer.Q THEN
		O10B_BDY_BOWL_ON_Q201_0:=1;
	END_IF
	IF Bowl_B_ON_Timer.Q THEN
		O10B_BDY_BOWL_ON_Q201_0:=0;
	END_IF
ELSE
	O10B_BDY_BOWL_ON_Q201_0:=1;	
END_IF

END_PROGRAM

// ---- POUs/Programs/OP20/OP20_MAIN.TcPOU
PROGRAM OP20_MAIN
VAR
	OP20_Modeselection_FB: Mode_Selection_Block1;
	Start: BOOL;
	Pause: BOOL;
	Gen_Timer: TON;
END_VAR

// Function Calling

OP20_Manual();
OP20_AUTOSEQUENCE();
OP20_Error();
OP20_Initialization_Seq();

//MOdeselection From HMI

IF (OP20_GVL.OP20_HMI_AutoMode AND NOT OP20_GVL.OP20_HMI_ManualMOde AND NOT OP20_GVL.OP20_HMI_StepMode) THEN
	OP20_Modeselection_FB.ModeWord:=1;
	ELSIF (NOT OP20_GVL.OP20_HMI_AutoMode AND OP20_GVL.OP20_HMI_ManualMOde AND NOT OP20_GVL.OP20_HMI_StepMode) THEN
		OP20_Modeselection_FB.ModeWord:=2;
	ELSIF  (NOT OP20_GVL.OP20_HMI_AutoMode AND NOT OP20_GVL.OP20_HMI_ManualMOde AND  OP20_GVL.OP20_HMI_StepMode) THEN
		OP20_Modeselection_FB.ModeWord:=3;
    ELSE   
		OP20_Modeselection_FB.ModeWord:=0;
END_IF
	
OP20_Safety_OK:=OperationEnable;

OP20_Modeselection_FB(
	ModeWord:= , 
	HomeConditionOK:=OP20_HomeConditionOK , 
	OperationEnable:=OP20_AutoSelected AND OP20_Safety_OK , 
	StartPB:=OP20_HMI_CycleStart , 
	SafetyAndNOError:= OP20_Safety_OK, 
	ModeAck:=TRUE , 
	HomingINProgress:=OP20_HomeRunning , 
	TempHomeOK:=OP20_Temp_hmeOK , 
	ResetPB:= , 
	AutoSelected=> OP20_AutoSelected, 
	ManualSelected=> OP20_ManualSelected, 
	StepSelected=>OP20_StepSelected , 
	ModeSelAck_Indication=> , 
	StatusDisplay=> , 
	AutoRunning:=OP20_AutoRunning, 
	StepRunning:=OP20_StepRunning , 
	StartEnable:=OP20_StartEnable  , 
	MachineStop:=OP20_Machine_Stop );


//IF (OP20_AutoSelected OR OP20_ManualSelected) AND ( NOT OP20_ErrorActive) AND OP20_Safety_OK THEN
//	SR20_Vert_servo.bEnable:=TRUE;
//ELSE
//	SR20_Vert_servo.bEnable:=FALSE;
//END_IF

IF OP20_Stop_Request AND NOT OP20_STN_ENABLE THEN
	OP20_Machine_Stop:=1;
END_IF
Gen_Timer(IN:=OP20_Machine_Stop,PT:=T#5S);
IF Gen_Timer.Q THEN
	OP20_Machine_Stop:=0;
END_IF

END_PROGRAM

// ---- FB/Mode_Selection_Block1.TcPOU
FUNCTION_BLOCK Mode_Selection_Block1
VAR_INPUT
	ModeWord 				:INT;
	HomeConditionOK 		:BOOL;
	OperationEnable 		:BOOL;
	StartPB 				:BOOL;
	SafetyAndNOError 		:BOOL;
	ModeAck 				:BOOL;
	HomingINProgress		:BOOL;
	TempHomeOK 				:BOOL;
	ResetPB 				:BOOL;
END_VAR
VAR_OUTPUT
	AutoSelected 			:BOOL;
	ManualSelected 			:BOOL;
	StepSelected 			:BOOL;
	ModeSelAck_Indication 	:BOOL;
	StatusDisplay 			:INT;
END_VAR
VAR_IN_OUT
	AutoRunning 			:BOOL;
	StepRunning 			:BOOL;
	StartEnable 			:BOOL;
	MachineStop 			:BOOL;
END_VAR
VAR
	CycleStart_PLS 					:Tc2_Standard.R_TRIG;
	CycleStart_Step_PLS				:Tc2_Standard.R_TRIG;
	Status 							:INT;
END_VAR



// Move Always "0" to the Status

Status := 0;


//Check Any Mode is Running

IF AutoRunning AND ModeWord <> 0 THEN Status := 1; END_IF
IF StepRunning AND ModeWord <> 0 THEN Status := 2; END_IF


// AutoMode Selected

IF ModeWord = 1 AND ModeAck AND Status = 0 THEN 
	 AutoSelected :=1;
	 ManualSelected :=0;
	 StepSelected :=0;
END_IF

 
// ManualMode Selected

IF ModeWord = 2 AND ModeAck AND Status = 0 AND NOT (AutoRunning OR StepRunning)THEN 
	 AutoSelected :=0;
	 ManualSelected :=1;
	 StepSelected :=0;
END_IF


// StepMode Selected

IF ModeWord = 3 AND ModeAck AND Status = 0 THEN 
	 AutoSelected :=0;
	 ManualSelected :=0;
	 StepSelected :=1;
END_IF


//Auto Running or Step Running

CycleStart_PLS(CLK := StartPB);

IF CycleStart_PLS.Q AND OperationEnable AND HomeConditionOK  AND SafetyAndNOError THEN
	IF AutoSelected THEN	
		AutoRunning := 1;
	END_IF
	IF StepSelected THEN	
		StepRunning := 1;
	END_IF
END_IF
 

// Start Enable

CycleStart_Step_PLS(CLK := StartPB);

IF (AutoRunning OR StepRunning AND CycleStart_Step_PLS.Q) AND OperationEnable AND SafetyAndNOError THEN
	StartEnable :=1;
ELSE 
	StartEnable :=0;
END_IF


// AutoRunning & StepRunning Reset

IF NOT OperationEnable OR NOT SafetyAndNOError OR MachineStop OR HomingINProgress THEN
	AutoRunning :=0;
	StepRunning :=0;
END_IF



					(*>>>>>>>>>>>>         Status Disply          <<<<<<<<<<<<*)


// Error Active Status Display

IF OperationEnable AND SafetyAndNOError THEN
	StatusDisplay :=1;
END_IF


// Mode Not Selected

IF SafetyAndNOError AND NOT MachineStop AND NOT ManualSelected AND NOT AutoSelected AND NOT StepSelected THEN
	StatusDisplay :=2;
END_IF


// Home Condition Not OK

IF SafetyAndNOError AND NOT MachineStop AND NOT HomeConditionOK AND NOT StartEnable AND (AutoSelected OR StepSelected) THEN
	StatusDisplay :=3;
END_IF


// Homing In Progress

IF SafetyAndNOError AND HomingINProgress AND NOT HomeConditionOK AND NOT StartEnable AND NOT MachineStop THEN
	StatusDisplay :=4;
END_IF


// Machine Forced Stop

IF SafetyAndNOError AND NOT StartEnable AND MachineStop THEN
	StatusDisplay :=5;
END_IF


// AutoRunning/StepRunning Status Display

IF SafetyAndNOError AND AutoRunning THEN
	StatusDisplay :=9;
END_IF


// StepRunning Status Display

IF SafetyAndNOError AND StepRunning THEN
	StatusDisplay :=10;
END_IF

END_FUNCTION_BLOCK

// ---- POUs/Programs/OP20/OP20_MANUAL.TcPOU
PROGRAM OP20_MANUAL
VAR

//	SR20_Vert_servo_ctrl:Servo_Control_1;
	SR20_Vert_servo_Axis :AXIS_REF;

	OP20_LH_OIL_SPIN_M: BOOL;
	OP20_RH_OIL_SPIN_M: BOOL;
	OP20_LH_OIL_SPRAY_M: BOOL;
	OP20_RH_OIL_SPRAY_M: BOOL;
	temp_safe: BOOL;
	temp:BOOL;
	temp_1: BOOL;

	
	error: BOOL;
	fb_initz: BOOL;
	SERVO_LIMIT_WARNING: BOOL;
	
	
	
	// COE READ PARAMETER 
	fbSdoRead  : FB_EcCoESdoRead;
    sNetId     : T_AmsNetId := '192.168.0.1.15.1';
    bExecute   : BOOL;
    nSlaveAddr : UINT := 1002;
    nIndex     : WORD := 16#1018;
    nSubIndex  : BYTE :=1;
    vendorId   : UDINT;
    bError     : BOOL;
    nErrId     : UDINT;
END_VAR


// IF MANUAL IS SELECTED 
IF ( MANUAL_SELECTED AND OP20_HMI_ManualMode )AND NOT ERROR_ACTIVE AND OperationEnable THEN
  
    IF OP20_LH_OIL_SPIN_M THEN
	    O20_LH_OIL_SPIN_ON_Q1150_1:=TRUE;
	ELSE 
		O20_LH_OIL_SPIN_ON_Q1150_1:=FALSE;
	END_IF
    IF OP20_RH_OIL_SPIN_M THEN
	    O20_RH_OIL_SPIN_ON_Q1150_3:=TRUE;
	ELSE 
		O20_RH_OIL_SPIN_ON_Q1150_3:=FALSE;
	END_IF	  
	IF OP20_LH_OIL_SPRAY_M THEN
	   O20_LH_OIL_DISPN_ON_Q1150_0:=TRUE;
	   O20_LH_OIL_DISPN_FRL_VLVE_ON_Q401_7:=1;
	ELSE 
	   O20_LH_OIL_DISPN_ON_Q1150_0:=0;
	   O20_LH_OIL_DISPN_FRL_VLVE_ON_Q401_7:=0;
	END_IF
	IF OP20_RH_OIL_SPRAY_M THEN
	   O20_RH_OIL_DISPN_ON_Q1150_2:=TRUE;
	   O20_RH_OIL_DISPN_FRL_VLVE_ON_Q401_5:=1;
	ELSE 
	   O20_RH_OIL_DISPN_ON_Q1150_2:=0;
	   O20_RH_OIL_DISPN_FRL_VLVE_ON_Q401_5:=0;
	END_IF	
	
END_IF

OP20_VERT_SERVO_POSITION := SR20_Vert_servo_ctrl.Actual_Position;
OP20_SERVO_POS_DONE	     := SR20_Vert_servo_ctrl.pos_done ;

OP20_VERT_SERVO_SFE_WRK_POS := OP20_HMI_Safe_Work;
OP20_VERT_SERVO_HME_POS     := OP20_HMI_Safe_Home;
OP20_VERT_SERVO_WRK_POS     := OP20_VERT_SERVO_WORK_POS;

IF In_Range(SR20_Vert_servo_status.actualPosition,OP20_VERT_SERVO_SFE_WRK_POS,1) THEN
	OP20_SERVO_ON_SFE_WRK := TRUE;
ELSE
	OP20_SERVO_ON_SFE_WRK := FALSE;
END_IF

IF In_Range(SR20_Vert_servo_status.actualPosition,OP20_VERT_SERVO_HME_POS,3) THEN
	OP20_SERVO_ON_HOME := TRUE;
ELSE
	OP20_SERVO_ON_HOME := FALSE;
END_IF

IF In_Range(SR20_Vert_servo_status.actualPosition,OP20_VERT_SERVO_WRK_POS,1) THEN
	OP20_SERVO_ON_WRK := TRUE;
ELSE
	OP20_SERVO_ON_WRK := FALSE;
END_IF	

SR20_Vert_servo(
	bAxis1_Ref_Switch:= , 
	bInit:= fb_initz, 
	bErrorReset:=OP20_HMI_Reset OR Servo_Reset , 
	bEnable:= Servo_Enable, 
	bMoveVelocity:= , 
	bHalt:= , 
	bManualMode:= MANUAL_SELECTED AND OP20_ManualSelected ,
	fHomePos:= , 
	fOverride:= , 
	fTargetPosition:=SR20_Vert_servo_ctrl.Position , 
	fTargetVelocity:=SR20_Vert_servo_ctrl.Velocity , 
	fAcc:= , 
	fDec:= ,
	Servo_High_Limit:= OP20_HMI_High_Limit,	
	Servo_Low_Limit:=  OP20_HMI_Low_Limit,	 	
	WARNING_LIMIT:=1,		
	Actual_Torque=> SR20_Vert_servo_ctrl.Actual_Torque ,
	Actual_position=>SR20_Vert_servo_ctrl.Actual_Position ,
    Actual_velocity=>SR20_Vert_servo_ctrl.Actual_Velocity ,
	TORQUE_LIMIT=>,	
	bmove_home:=SR20_Vert_servo_ctrl.Axis_Home_Cmd ,
	baxis_in_home_pos=>SR20_Vert_servo_ctrl.Axis_In_Home ,
	Safe_move_Conditions:=Servo_Safety,
	Axis:= SR20_Vert_servo_Axis , 
	bHome:=SR20_Vert_servo_ctrl.Bsethome ,
	HME_WRITE_ADD:= 16#5001, 
    bSetPosition:=SR20_Vert_servo_ctrl.Bsetpos , 
	bMoveAbsolute:=SR20_Vert_servo_ctrl.ABSmove_Start ,
	bMoveRelative:=SR20_Vert_servo_ctrl.RELmove_Start , 
	bMoveTorque :=SR20_Vert_servo_ctrl.Torque_mode_Start,
	stManualModeAxis:=SR20_Vert_servo_status , 
	sAxisState=>SR20_Vert_servo_ctrl.Axis_State , 
	bAxis_ready=>SR20_Vert_servo_ctrl.Axis_ready , 
	bAxisInPosition=> SR20_Vert_servo_ctrl.Axis_In_Pos, 
	bAxisError=>SR20_Vert_servo_ctrl.Axis_Error , 
	bAxisEnabled=> SR20_Vert_servo_ctrl.Axis_Enabled, 
	bAxisHomed=> SR20_Vert_servo_ctrl.Axis_reference,
	bTorqueReached=> SR20_Vert_servo_ctrl.Trq_reached, 
	bSetPositionDone=>   ,
	bsafe_to_move=> ,
	bABS_Pos_done=> SR20_Vert_servo_ctrl.pos_done , 
	bHaltDone=> ,
	SERVO_LIMIT_WARNING=>SERVO_LIMIT_WARNING, 
	bSTOPDone=> , 
	bHomeDone=> , 
	bDone=> );	
	
IF OP20_ManualSelected AND MANUAL_SELECTED THEN
	SR20_Vert_servo_status.targetVelocity:=50;
END_IF


//COE READ OP 20 VERTICLE MOTOR TEMPERATURE
fbSdoRead(sNetId:= sNetId,nSlaveAddr :=nSlaveAddr, nIndex:=nIndex,
		 nSubIndex :=nSubIndex, pDstBuf:= ADR(vendorId), 
		 cbBufLen:=SIZEOF(vendorId),bExecute:=bExecute);
		 bError:=fbSdoRead.bError;
		 nErrId:=fbSdoRead.nErrId;

END_PROGRAM

// ---- POUs/Programs/OP20/OP20_AUTOSEQUENCE.TcPOU
PROGRAM OP20_AUTOSEQUENCE
VAR	
//BOOL
	OP20_STN_ERR					: BOOL;
	OP20_LH_A_OIL_Dispense			: BOOL;
	OP20_RH_A_OIL_Dispense			: BOOL;
	OP20_RH_A_OIL_SPIN 				: BOOL;
	OP20_LH_A_OIL_SPIN				: BOOL;
	OP20_Oil_Range					: BOOL;

//TON
	OP20_Oiling_Timer				: TON;
	MOVER_POS_RECHED_R				: R_trig;
	OP20_STN_MOVER: INT;
	Dry_Run : BOOL;
	OP20_Cycle_Time_FB : FB_Cycletime;	
	OP20_WRK_DELAY : TON;
	WRK_DELAY	: INT :=500;

END_VAR

IF OP20_AutoSelected AND NOT OP20_ErrorActive AND OperationEnable THEN
    SR20_Vert_servo_ctrl.Velocity := OP20_HMI_Servo_Speed;
	O20_LH_OIL_DISPN_ON_Q1150_0:=TRUE ;
	O20_RH_OIL_DISPN_ON_Q1150_2:=TRUE ;
	O20_LH_OIL_DISPN_FRL_VLVE_ON_Q401_7:=OP20_LH_A_OIL_Dispense;
	O20_RH_OIL_DISPN_FRL_VLVE_ON_Q401_5:=OP20_RH_A_OIL_Dispense;
	O20_LH_OIL_SPIN_ON_Q1150_1:=OP20_RH_A_OIL_SPIN ;
	O20_RH_OIL_SPIN_ON_Q1150_3:=OP20_LH_A_OIL_SPIN;
END_IF

OP20_OIL_TIMER:=OP20_OIL_TIMER; //OP20_DLY_OIL_ON;
// AUTO MODE
IF (NOT OP20_AutoSelected OR OP20_ErrorActive OR OP20_HomeRunning OR NOT  OperationEnable ) THEN
	OP20_AutoRunning:= FALSE;
	OP20_AutoSeq:= 10;
	OP20_STN_ENABLE:=FALSE;
	OP20_STN_RUNNING:=FALSE;
END_IF	
		
IF (OP20_ErrorActive OR OP20_HomeRunning OR NOT OperationEnable) THEN
	O20_LH_OIL_DISPN_ON_Q1150_0 :=0;
	O20_RH_OIL_DISPN_ON_Q1150_2 :=0;
	O20_LH_OIL_SPIN_ON_Q1150_1  :=0;
	O20_RH_OIL_SPIN_ON_Q1150_3  :=0;
END_IF	
																							
CASE OP20_AutoSeq OF
		
		10: IF (OP20_AutoSelected) THEN		// Check Automode Selected
				OP20_AutoSeq:=20;
	        END_IF
		
	    20:IF ( NOT OP20_ErrorActive) THEN		//Check No error
		       OP20_AutoSeq:=30;
      	   END_IF
		   
      	30:IF (NOT OP20_HomeRunning) THEN		//Check No Homerunning
      		   OP20_AutoSeq :=40;
      	   END_IF
		   
        40:IF (OP20_Main.OP20_Modeselection_FB.TempHomeOK)THEN	//Check Machine in Home
      		   OP20_AutoSeq:= 50;
      	   END_IF
		   
      	50:IF ( OP20_STN_ENABLE AND OP20_STN_RUNNING ) THEN		// Check Operation Completed Reset
      		   OP20_AutoSeq:=70;
		   ELSE
	   		   OP20_AutoSeq:=60;
      	   END_IF
		   
	   60:IF  (AUTO_RUNNING OR (NOT AUTO_RUNNING AND OP20_HMI_CycleStart)) THEN		//Machine Start in Fully Automatic or Press Cycle Start For Semi Automatic
		    OP20_HomeConditionOK:=TRUE;
	 			IF( OP20_Main.OP20_Modeselection_FB.HomeConditionOK AND OP20_AutoSelected) THEN
					OP20_AutoRunning:=TRUE;
					OP20_StepRunning:= FALSE;
				
				ELSIF (OP20_Main.OP20_Modeselection_FB.HomeConditionOK AND OP20_StepSelected) THEN
					OP20_AutoRunning:=FALSE;
					OP20_StepRunning:= TRUE;
				END_IF;
		  END_IF
		   IF ((OP20_AutoRunning OR OP20_StepRunning) AND OP20_StartEnable) THEN
				OP20_AutoSeq:= 70;
		   END_IF

      	70:  // SERVO POSITION SAFE CHECK
	       IF (OP20_SERVO_ON_SFE_WRK OR OP20_SERVO_ON_HOME)AND OP20_SERVO_POS_DONE AND NOT SR20_Vert_servo_ctrl.ABSmove_Start THEN 
	         SR20_Vert_servo_ctrl.Position := OP20_VERT_SERVO_WRK_POS;
			 IF SR20_Vert_servo_ctrl.Position=OP20_VERT_SERVO_WRK_POS THEN
 				OP20_AutoSeq:=75;
			 END_IF	
	       END_IF
			   
		75: // WAITING FOR MOVER AND MOVING SERVO TO TARGET POSITION
			IF OP20_STN_ENABLE THEN
			 	SR20_Vert_servo_ctrl.ABSmove_Start:=TRUE;
			 	OP20_STN_RUNNING :=1;
			 	OP20_LH_OIL_OK:=FALSE;
			 	OP20_RH_OIL_OK:=FALSE;
			 	OP20_AutoSeq:=80;
			END_IF
			
		80: // START THE SPINNER OK COMPONENT FIXTURE	 
			 IF OP20_FIXTURE_1=10 AND OP20_FIXTURE_2<>10  THEN
			   OP20_LH_A_OIL_Dispense:=1;
			   OP20_AutoSeq:=100;			   
			 ELSIF OP20_FIXTURE_2=10 AND OP20_FIXTURE_1<>10 THEN
			   OP20_RH_A_OIL_Dispense:=1;
			   OP20_AutoSeq:=100;			   
			 ELSIF OP20_FIXTURE_1=10 AND OP20_FIXTURE_2=10 THEN  
				OP20_LH_A_OIL_Dispense:=1;
				OP20_RH_A_OIL_Dispense:=1;
			    OP20_AutoSeq:=100;				
			ELSIF OP20_FIXTURE_1<>10 AND OP20_FIXTURE_2<>10 THEN
			 	OP20_AutoSeq:=120;	
			END_IF
	  
		100: //START THE OILLING UNIT 
		     	IF OP20_Oiling_Timer.Q AND OP20_FIXTURE_1=10 AND OP20_FIXTURE_2=10 THEN
					OP20_LH_OIL_OK:=TRUE;
					OP20_RH_OIL_OK:=TRUE;
					OP20_AutoSeq:=120;	
			 	ELSIF OP20_Oiling_Timer.Q AND OP20_FIXTURE_1=10 THEN
					OP20_LH_OIL_OK:=TRUE;	
					OP20_AutoSeq:=120;	
			 	ELSIF OP20_Oiling_Timer.Q AND OP20_FIXTURE_2=10 THEN
					OP20_RH_OIL_OK:=TRUE;
					OP20_AutoSeq:=120;	
		     	END_IF
				
			 				
		120:    IF OP20_SERVO_ON_WRK AND (OP20_LH_OIL_OK OR OP20_RH_OIL_OK) THEN
					OP20_RH_A_OIL_SPIN:=1;
		            OP20_LH_A_OIL_SPIN:=1;
				END_IF
				SR20_Vert_servo_ctrl.Position:=OP20_VERT_SERVO_SFE_WRK_POS;
				IF OP20_LH_OIL_OK THEN
					MOVER_CMP_STATUS[OP20_STN_MOVER][1]	:=20;
				ELSE
					MOVER_CMP_STATUS[OP20_STN_MOVER][1]	:=20;				
				END_IF
				IF OP20_RH_OIL_OK THEN
					MOVER_CMP_STATUS[OP20_STN_MOVER][2]	:=20;
				ELSE                                 
					MOVER_CMP_STATUS[OP20_STN_MOVER][2]	:=20;				
				END_IF	
				IF OP20_WRK_DELAY.Q THEN
					OP20_AutoSeq:=140;		
				END_IF	
			
		140:  IF NOT SR20_Vert_servo_ctrl.ABSmove_Start AND OP20_SERVO_ON_WRK  THEN			 			 
			   SR20_Vert_servo_ctrl.ABSmove_Start:=TRUE;
			   OP20_AutoSeq:=160;
			 END_IF				  
	     	  	  	
		160: // SERVO DONE AND RESET THE DONE BITS
			IF NOT In_Range(SR20_Vert_servo_status.actualPosition,OP20_VERT_SERVO_WRK_POS,Oil_Region) THEN
					OP20_RH_A_OIL_SPIN:=0;
		            OP20_LH_A_OIL_SPIN:=0;				
			END_IF
			IF NOT SR20_Vert_servo_ctrl.ABSmove_Start AND OP20_SERVO_ON_SFE_WRK THEN
			  SR20_Vert_servo_ctrl.ABSmove_Start:=FALSE;
			  OP20_STN_ENABLE	:=0;
			  OP20_STN_RUNNING  :=0;
			  IF (MOVER_CMP_STATUS[OP20_STN_MOVER][1]=21) AND (MOVER_CMP_STATUS[OP20_STN_MOVER][1]=21) THEN
					MOVER_STP_NO[OP20_STN_MOVER]	:= (OP160_XTS_POS_NO*10);
				ELSE
				STATION_DONE[OP20_STN_MOVER][OP20_XTS_POS_NO]			:= TRUE;					
			  END_IF
	
			  OP20_AutoSeq:=70;			
			END_IF

END_CASE	

OP20_Cycle_Time_FB(i_b_startTime:=OP20_STN_ENABLE , i_b_stopTime:= NOT OP20_STN_ENABLE , o_t_StationTime=>OP20_Cycle_time );					


OP20_WRK_DELAY(IN:=OP20_SERVO_ON_WRK,PT:=INT_TO_TIME(WRK_DELAY));

Dry_Run:=All_Station_Dry_Run;

IF Dry_Run THEN
	OP20_FIXTURE_1:=10;
	OP20_FIXTURE_2:=10;
ELSE 
	OP20_FIXTURE_1:=MOVER_CMP_STATUS[OP20_STN_MOVER][1];
	OP20_FIXTURE_2:=MOVER_CMP_STATUS[OP20_STN_MOVER][2];	
END_IF

//Timers
OP20_Oiling_Timer(IN:=OP20_LH_A_OIL_Dispense OR OP20_RH_A_OIL_Dispense, PT:=INT_TO_TIME(OP20_OIL_TIMER));
IF OP20_Oiling_Timer.Q THEN
	OP20_LH_A_OIL_Dispense:=0;
	OP20_RH_A_OIL_Dispense:=0;
END_IF				
////################################ STATION ENABLE CONTION    ############################

	OP20_STN_MOVER					:= MOVER_POSITION[OP20_XTS_POS_NO];
	IF AUTO_WITH_XTS THEN
	IF OP20_STN_MOVER>0 THEN
	IF NOT(END_OF_CYCLE AND MOVER_CMP_STATUS[OP20_STN_MOVER][1]=5 AND MOVER_CMP_STATUS[OP20_STN_MOVER][2]=5)THEN
	OP20_STN_ENABLE					:= MOVER_POS_RECHED[OP20_STN_MOVER] AND ((MOVER_CMP_STATUS[OP20_STN_MOVER][1]=10)OR
											(MOVER_CMP_STATUS[OP20_STN_MOVER][2]=10)) AND STATION_ENABLE_CONTROL;
	ELSE
	STATION_DONE[OP20_STN_MOVER][OP20_XTS_POS_NO]			:= TRUE;		
	END_IF
	ELSE
	OP20_STN_ENABLE										:= FALSE;
	END_IF
	END_IF

END_PROGRAM

// ---- FB/FB_cycleTime.TcPOU
FUNCTION_BLOCK FB_cycleTime
VAR_INPUT
i_b_startTime			:BOOL;
i_b_stopTime			:BOOL;
END_VAR
VAR_OUTPUT
o_t_StationTime			: UDINT;	
END_VAR

VAR
startTime				: ULINT;
stopTime				: ULINT;
FPstart					: BOOL;
FPstop					: BOOL;
HMFPstart				: BOOL;
HMFPstop				: BOOL;	
END_VAR

FPstart:= i_b_startTime AND NOT HMFPstart;
HMFPstart:= i_b_startTime;
	
	
FPstop:= i_b_stopTime AND NOT HMFPstop;
HMFPstop:= i_b_stopTime;


IF FPstart THEN
	startTime:= F_GetSystemTime();
END_IF

IF FPstop THEN
	stopTime:= F_GetSystemTime();
	o_t_StationTime:= ULINT_TO_UDINT(stopTime-startTime)/10000;
END_IF

END_FUNCTION_BLOCK

// ---- POUs/Programs/OP20/OP20_ERROR.TcPOU
PROGRAM OP20_ERROR
VAR
	OP20_StErr_1: TON;
	OP20_Step_Err_2: TON;
	OP20_StepErr_3: TON;
	OP20_StErr_4: TON;
	OP20_Step_Err_5: TON;
	OP20_StepErr_6: TON;
//	end: INT;
END_VAR


//Reset ErrorActive
IF (OP20_HMI_Reset OR Servo_Reset) THEN 
	OP20_GVL.OP20_ErrorActive:= FALSE;
	OP20_GVL.OP20_ErrorWord_0:= 0;
	OP20_GVL.OP20_ErrorWord_1:= 0;
	OP20_GVL.OP20_ErrorWord_2:= 0;	
END_IF

//(OP20_GVL.OP20_ErrorWord_0<>0) OR
// Set ERROR ACTIVE
IF ( (OP20_GVL.OP20_ErrorWord_1<>0) OR (OP20_GVL.OP20_ErrorWord_2<>0)) THEN
	OP20_GVL.OP20_ErrorActive:= TRUE;
END_IF


OP20_ErrorWord_0.0:= SR20_Vert_servo_ctrl.Axis_Error;
OP20_ErrorWord_0.1:= NOT OperationEnable;
// Auto Seq Step Error
//Servo not reaching work position
OP20_StErr_1(IN:=(OP20_GVL.OP20_AUTO_STP_NO=80) , PT:=T#5S , Q=> , ET=> );
IF (OP20_GVL.OP20_AUTO_STP_NO=80 AND NOT OP20_GVL.OP20_SERVO_ON_WRK AND OP20_StErr_1.Q) THEN
	OP20_GVL.OP20_ErrorWord_0.2:=TRUE;
END_IF

// Servo Not Reached home position or safe-work position
OP20_Step_Err_2(IN:=OP20_GVL.OP20_AUTO_STP_NO=160, PT:=T#5S , Q=> , ET=> );
IF (OP20_GVL.OP20_AUTO_STP_NO=160 AND NOT OP20_SERVO_ON_SFE_WRK AND OP20_Step_Err_2.Q) THEN
	OP20_GVL.OP20_ErrorWord_0.3:=TRUE;
END_IF
OP20_GVL.OP20_ErrorWord_0.4:=0;
//OP20_StepErr_3(IN:=( OP20_HomeRunning AND (OP20_Homing_Seq=10) AND NOT SR20_Vert_servo_ctrl.Axis_In_Home), PT:=T#10S , Q=> , ET=> );
//IF OP20_StepErr_3.Q THEN
//	OP20_GVL.OP20_ErrorWord_0.4:=TRUE;
//END_IF

END_PROGRAM

// ---- POUs/Programs/OP20/OP20_Initialization_Seq.TcPOU
PROGRAM OP20_Initialization_Seq
VAR
END_VAR

IF (SR20_Vert_servo_ctrl.Axis_In_Home)THEN
OP20_Temp_hmeOK:=TRUE;
OP20_HomeRunning:=FALSE;
OP20_Homing_Seq:=0;
ELSE
	OP20_Temp_hmeOK:=FALSE;	
END_IF

CASE OP20_Homing_Seq OF
	0: IF (OP20_AutoSelected AND NOT OP20_HomeRunning AND NOT OP20_ErrorActive AND NOT OP20_AutoRunning AND NOT OP20_StepRunning AND NOT OP20_Temp_hmeOK) THEN
		OP20_HomeRunning:=TRUE;
		OP20_Homing_Seq:=10;	
	   END_IF
	10:IF (OP20_HomeRunning AND (OP20_HMI_Homing OR HMI_Reset))THEN 
			IF (SR20_Vert_servo_ctrl.Axis_In_Home) THEN 
				//OP20_Homing_Seq:=20;
				SR20_Vert_servo_ctrl.Axis_Home_Cmd:=FALSE;
			ELSE
				SR20_Vert_servo_ctrl.Position:=0;
				SR20_Vert_servo_ctrl.Velocity:=100;
				SR20_Vert_servo_ctrl.ABSmove_Start:=TRUE;
				SR20_Vert_servo_ctrl.Axis_Home_Cmd:=TRUE;
	    	END_IF
			IF SR20_Vert_servo_ctrl.Axis_In_Home THEN
			  OP20_Homing_Seq:=20;			
			END_IF
	   END_IF		
	20:	OP20_Homing_Seq:=0;
		OP20_HomeRunning:=FALSE;
		OP20_HMI_Homing:=FALSE;
END_CASE

END_PROGRAM

// ---- POUs/Programs/OP30/OP30_MAIN.TcPOU
PROGRAM OP30_MAIN
VAR
	OP30_Modeselection_FB: Mode_Selection_Block1;
	TP_100ms: TP;
	Pulse_1s: BOOL;
	Times: LREAL;
	Pge_NUM : INT;
	Gen_Timer	: TON;
END_VAR


OP30_Manual();
OP30_AUTOSEQUENCE();
OP30_Conveyor_Cam_Seq();
OP30_Error();
OP30_Initialize_Seq();
OP30_Camera_FB();

//MOdeselection From HMI

IF (OP30_GVL.OP30_HMI_AutoMode AND NOT OP30_GVL.OP30_HMI_ManualMOde AND NOT OP30_GVL.OP30_HMI_StepMode) THEN
	OP30_Modeselection_FB.ModeWord:=1;
	ELSIF (NOT OP30_GVL.OP30_HMI_AutoMode AND OP30_GVL.OP30_HMI_ManualMOde AND NOT OP30_GVL.OP30_HMI_StepMode) THEN
		OP30_Modeselection_FB.ModeWord:=2;
	ELSIF  (NOT OP30_GVL.OP30_HMI_AutoMode AND NOT OP30_GVL.OP30_HMI_ManualMOde AND  OP30_GVL.OP30_HMI_StepMode) THEN
		OP30_Modeselection_FB.ModeWord:=3;
    ELSE   
		OP30_Modeselection_FB.ModeWord:=0;
END_IF

(*IF  (OP30_AutoSelected OR OP30_ManualSelected ) AND NOT OP30_ErrorActive AND OP30_Safety_OK THEN
  SR30_CONV_servo.bEnable:=TRUE;
  SR30_HORI_servo.bEnable:=TRUE;
  SR30_VERT_servo.bEnable:=TRUE;
ELSE 
  SR30_CONV_servo.bEnable:=FALSE;
  SR30_HORI_servo.bEnable:=FALSE;
  SR30_VERT_servo.bEnable:=FALSE;	
END_IF*)
(*
IF SR30_CONV_servo.bAxisError OR SR30_HORI_servo.bAxisError OR SR30_VERT_servo.bAxisError THEN
	OP30_ErrorActive:=TRUE;
END_IF*)
	
OP30_Modeselection_FB(
	ModeWord:= , 
	HomeConditionOK:=OP30_HomeConditionOK , 
	OperationEnable:=OP30_AutoSelected AND OP30_Safety_OK , 
	StartPB:=OP30_HMI_Cycle_Start , 
	SafetyAndNOError:= OP30_Safety_OK, 
	ModeAck:=TRUE , 
	HomingINProgress:=OP30_HomeRunning , 
	TempHomeOK:=OP30_Temp_hmeOK , 
	ResetPB:= , 
	AutoSelected=> OP30_AutoSelected, 
	ManualSelected=> OP30_ManualSelected, 
	StepSelected=>OP30_StepSelected , 
	ModeSelAck_Indication=> , 
	StatusDisplay=> , 
	AutoRunning:=OP30_AutoRunning, 
	StepRunning:=OP30_StepRunning , 
	StartEnable:=OP30_StartEnable  , 
	MachineStop:=OP30_Machine_Stop );
		
OP30_Safety_OK:=OperationEnable;	

IF OP30_Stop_Request AND NOT OP30_STN_ENABLE THEN
	OP30_Machine_Stop:=1;
END_IF
Gen_Timer(IN:=OP30_Machine_Stop,PT:=T#5S);
IF Gen_Timer.Q THEN
	OP30_Machine_Stop:=0;
END_IF

END_PROGRAM

// ---- FB/Pulse_1s.TcPOU
FUNCTION_BLOCK Pulse_1s
VAR_INPUT
END_VAR
VAR_OUTPUT
END_VAR
VAR
	T1: TON;
	T2: TON;
	Out:bool;
	ON: BOOL;
	Sec: R_TRIG;
	Count: INT;
	Check: TON;
	total: TIME;
END_VAR

//Check(IN:=STart , PT:=T#10S , Q=> , ET=>total );
IF (ON AND NOT Check.q) THEN
	
T1(IN:= NOT T2.q , PT:= T#50MS, Q=> , ET=> );
T2(IN:=T1.q , PT:=T#50MS , Q=> , ET=> );
END_IF 
//IF ( T2.q) THEN
//	Out:=TRUE;
//	ELSE
//		Out:=FALSE;
//	END_IF
Sec(CLK:= T1.q , Q=> );
IF MAIN.temp THEN
	Count:=Count+1;
END_IF
//IF NOT On THEN
	//Count:=0;
//END_IF

END_FUNCTION_BLOCK

// ---- POUs/Programs/OP30/OP30_MANUAL.TcPOU
PROGRAM OP30_MANUAL
VAR

	SR30_Vert_servo_Axis :AXIS_REF;
	SR30_Hori_servo_Axis :AXIS_REF;
	SR30_Conv_servo_Axis :AXIS_REF;
	SR30_GUIDE_GRP_AXIS	 :AXIS_REF;
	LH_Gripper_bMove	 : BOOL;
	RH_Gripper_bMove	 : BOOL;
	temp_safe: BOOL;
	temp:BOOL;
	error30: BOOL;
	OP30Enable: BOOL;
	FESTO_NOT_NEED: BOOL;
	NOT_REQ: BOOL;
	Gripper_Ref_Timer : TON;
	temp30: BOOL;
	Test : TON;
	Grip_Test : INT;

END_VAR


OP30_VERT_SERVO_POSITION    := SR30_Vert_servo_ctrl.Actual_Position;
OP30_VERT_SERVO_POS_DONE	:= SR30_Vert_servo_ctrl.pos_done ;

OP30_HORI_SERVO_POSITION    := SR30_Hori_servo_ctrl.Actual_Position;
OP30_HORI_SERVO_POS_DONE	:= SR30_Hori_servo_ctrl.pos_done ;

OP30_CONV_SERVO_POSITION    := SR30_CONV_servo_ctrl.Actual_Position;
OP30_CONV_SERVO_POS_DONE	:= SR30_CONV_servo_ctrl.pos_done ;


// VERTICAL SERVO 
IF In_Range(SR30_Vert_servo_status.actualPosition,OP30_VERT_SERVO_SFE_WRK_POS,1) THEN
	OP30_VERT_SERVO_ON_SFE_WRK := TRUE;
ELSE
	OP30_VERT_SERVO_ON_SFE_WRK := FALSE;
END_IF

IF In_Range(SR30_Vert_servo_status.actualPosition,OP30_VERT_SERVO_HME_POS,3) THEN
	OP30_VERT_SERVO_ON_HOME := TRUE;
ELSE
	OP30_VERT_SERVO_ON_HOME := FALSE;
END_IF

IF In_Range(SR30_Vert_servo_status.actualPosition,OP30_VERT_SERVO_PICK_POS,3) THEN
	OP30_VERT_SERVO_ON_WRK_PICK := TRUE;
ELSE
	OP30_VERT_SERVO_ON_WRK_PICK := FALSE;
END_IF		

IF In_Range(SR30_Vert_servo_status.actualPosition,OP30_VERT_SERVO_PLACE_POS,3) THEN
	OP30_VERT_SERVO_ON_WRK_PLACE := TRUE;
ELSE
	OP30_VERT_SERVO_ON_WRK_PLACE := FALSE;
END_IF

//HORIZONTAL SERVO
IF In_Range(SR30_Hori_servo_status.actualPosition,OP30_HORI_SERVO_SFE_WRK_POS,1) THEN
	OP30_HORI_SERVO_ON_SFE_WRK := TRUE;
ELSE
	OP30_HORI_SERVO_ON_SFE_WRK := FALSE;
END_IF

IF In_Range(SR30_Hori_servo_status.actualPosition,OP30_HORI_SERVO_HME_POS,2) THEN
	OP30_HORI_SERVO_ON_HOME := TRUE;
ELSE
	OP30_HORI_SERVO_ON_HOME := FALSE;
END_IF

IF In_Range(SR30_Hori_servo_status.actualPosition,OP30_HORI_SERVO_SAFE_PICK_POS,1) THEN
	OP30_HORI_SERVO_ON_SFE_WRK_PICK := TRUE;
ELSE
	OP30_HORI_SERVO_ON_SFE_WRK_PICK := FALSE;
END_IF	

IF In_Range(SR30_Hori_servo_status.actualPosition,OP30_HORI_SERVO_PICK_POS,4) THEN
	OP30_HORI_SERVO_ON_WRK_PICK := TRUE;
ELSE
	OP30_HORI_SERVO_ON_WRK_PICK := FALSE;
END_IF	

IF In_Range(SR30_Hori_servo_status.actualPosition,OP30_HORI_SERVO_PLACE_POS,1) THEN
	OP30_HORI_SERVO_ON_WRK_PLACE := TRUE;
ELSE
	OP30_HORI_SERVO_ON_WRK_PLACE := FALSE;
END_IF	

//CONVEYOR SERVO

IF In_Range(SR30_CONV_servo_status.actualPosition,OP30_CONV_SERVO_SFE_WRK_POS,1) THEN
	OP30_CONV_SERVO_ON_SFE_WRK := TRUE;
ELSE
	OP30_CONV_SERVO_ON_SFE_WRK := FALSE;
END_IF

IF In_Range(SR30_CONV_servo_status.actualPosition,OP30_CONV_SERVO_HME_POS,1) THEN
	OP30_CONV_SERVO_ON_HOME := TRUE;
ELSE
	OP30_CONV_SERVO_ON_HOME := FALSE;
END_IF

IF In_Range(SR30_CONV_servo_status.actualPosition,OP30_CONV_SERVO_WRK_POS,1) THEN
	OP30_CONV_SERVO_ON_WRK := TRUE;
ELSE
	OP30_CONV_SERVO_ON_WRK := FALSE;
END_IF	




OP30_GVL.SR30_Vert_servo(
	bAxis1_Ref_Switch:= temp, 
	bInit:= , 
	bErrorReset:=OP30_HMI_Reset OR Servo_Reset , 
	bEnable:=Servo_Enable, 
	bMoveVelocity:= , 
	bHalt:= , 
	bManualMode:= OP30_ManualSelected AND MANUAL_SELECTED ,
	fHomePos:= , 
	fOverride:= , 
	fTargetPosition:=SR30_Vert_servo_ctrl.Position , 
	fTargetVelocity:=SR30_Vert_servo_ctrl.Velocity , 
	fAcc:= , 
	fDec:= ,
	Servo_High_Limit:= OP30_HMI_Vert_High_Limit,	
	Servo_Low_Limit:=  OP30_HMI_Vert_Low_Limit,	 	
	WARNING_LIMIT:=     1,		
	Actual_Torque=> SR30_Vert_servo_ctrl.Actual_Torque ,
	Actual_position=>SR30_Vert_servo_ctrl.Actual_Position ,
    Actual_velocity=>SR30_Vert_servo_ctrl.Actual_Velocity ,	
	bmove_home:=SR30_Vert_servo_ctrl.Axis_Home_Cmd ,
	baxis_in_home_pos=>SR30_Vert_servo_ctrl.Axis_In_Home ,
	Safe_move_Conditions:= Servo_Safety ,
	HME_WRITE_ADD:= 16#5006,
	Axis:= SR30_Vert_servo_Axis , 
	bHome:=SR30_Vert_servo_ctrl.Bsethome , 
    bSetPosition:=SR30_Vert_servo_ctrl.Bsetpos , 
	bMoveAbsolute:=SR30_Vert_servo_ctrl.ABSmove_Start , 
	bMoveRelative:=SR30_Vert_servo_ctrl.RELmove_Start , 
	bMoveTorque :=SR30_Vert_servo_ctrl.Torque_mode_Start,
	stManualModeAxis:=SR30_Vert_servo_status , 
	sAxisState=>SR30_Vert_servo_ctrl.Axis_State , 
	bAxis_ready=>SR30_Vert_servo_ctrl.Axis_ready , 
	bAxisInPosition=> SR30_Vert_servo_ctrl.Axis_In_Pos, 
	bAxisError=>SR30_Vert_servo_ctrl.Axis_Error , 
	bAxisEnabled=> SR30_Vert_servo_ctrl.Axis_Enabled, 
	bAxisHomed=> SR30_Vert_servo_ctrl.Axis_reference,
	bTorqueReached=> SR30_Vert_servo_ctrl.Trq_reached, 
	bSetPositionDone=>   ,
	bsafe_to_move=> ,
	bABS_Pos_done=> SR30_Vert_servo_ctrl.pos_done , 
	bHaltDone=> , 
	bSTOPDone=> , 
	bHomeDone=> , 
	bDone=> );	

OP30_GVL.SR30_HORI_servo(
	bAxis1_Ref_Switch:= , 
	bInit:= , 
	bErrorReset:=OP30_HMI_Reset OR Servo_Reset , 
	bEnable:= Servo_Enable , 
	bMoveVelocity:= , 
	bHalt:= , 
	bManualMode:= OP30_ManualSelected AND MANUAL_SELECTED ,
	fHomePos:= , 
	fOverride:= , 
	fTargetPosition:= SR30_HORI_servo_ctrl.Position , 
	fTargetVelocity:= SR30_HORI_servo_ctrl.Velocity, 
	fAcc:= , 
	fDec:= ,
	Servo_High_Limit:= OP30_HMI_Hori_High_Limit,	
	Servo_Low_Limit:= OP30_HMI_Hori_Low_Limit,	 	
	WARNING_LIMIT:=1,		
	Actual_Torque=> SR30_HORI_servo_ctrl.Actual_Torque ,
	Actual_position=>SR30_HORI_servo_ctrl.Actual_Position ,
    Actual_velocity=>SR30_HORI_servo_ctrl.Actual_Velocity ,	
	bmove_home:=SR30_HORI_servo_ctrl.Axis_Home_Cmd ,
	baxis_in_home_pos=>SR30_HORI_servo_ctrl.Axis_In_Home ,
	Safe_move_Conditions:=Servo_Safety,
	HME_WRITE_ADD:= 16#5005,
	Axis:= SR30_HORI_servo_Axis , 
	bHome:=SR30_HORI_servo_ctrl.Bsethome , 
    bSetPosition:=SR30_HORI_servo_ctrl.Bsetpos , 
	bMoveAbsolute:=SR30_HORI_servo_ctrl.ABSmove_Start , 
	bMoveRelative:=SR30_HORI_servo_ctrl.RELmove_Start , 
	bMoveTorque :=SR30_HORI_servo_ctrl.Torque_mode_Start,
	stManualModeAxis:=SR30_HORI_servo_status , 
	sAxisState=>SR30_HORI_servo_ctrl.Axis_State , 
	bAxis_ready=>SR30_HORI_servo_ctrl.Axis_ready , 
	bAxisInPosition=> SR30_HORI_servo_ctrl.Axis_In_Pos, 
	bAxisError=>SR30_HORI_servo_ctrl.Axis_Error , 
	bAxisEnabled=> SR30_HORI_servo_ctrl.Axis_Enabled, 
	bAxisHomed=> SR30_HORI_servo_ctrl.Axis_reference,
	bTorqueReached=> SR30_HORI_servo_ctrl.Trq_reached, 
	bSetPositionDone=>   ,
	bsafe_to_move=> ,
	bABS_Pos_done=> SR30_HORI_servo_ctrl.pos_done , 
	bHaltDone=> , 
	bSTOPDone=> , 
	bHomeDone=> , 
	bDone=> );

OP30_GVL.SR30_CONV_servo(
	bAxis1_Ref_Switch:= temp, 
	bInit:= , 
	bErrorReset:=OP30_HMI_Reset OR Servo_Reset , 
	bEnable:=Servo_Enable, 
	bMoveVelocity:=SR30_CONV_servo_ctrl.VELmove_Start , 
	bHalt:= , 
	bManualMode:= OP30_ManualSelected AND MANUAL_SELECTED,
	fHomePos:= , 
	fOverride:= , 
	fTargetPosition:= SR30_CONV_servo_ctrl.Position, 
	fTargetVelocity:= SR30_CONV_servo_ctrl.Velocity,
	LIMIT_BYPASS:=1, 
	fAcc:= , 
	fDec:= ,
	Actual_Torque=> SR30_CONV_servo_ctrl.Actual_Torque ,
	Actual_position=>SR30_CONV_servo_ctrl.Actual_Position ,
    Actual_velocity=>SR30_CONV_servo_ctrl.Actual_Velocity ,
	POS_TORQUE_LIMIT=>,
	NEG_TORQUE_LIMIT=>,
	bmove_home:=SR30_CONV_servo_ctrl.Axis_Home_Cmd ,
	baxis_in_home_pos=>SR30_CONV_servo_ctrl.Axis_In_Home ,
	Safe_move_Conditions:=Servo_Safety,
	Axis:= SR30_CONV_servo_Axis ,
	HME_WRITE_ADD:= 16#5007,
	Torque_limit_perent:=,
	bHome:=SR30_CONV_servo_ctrl.Bsethome , 
    bSetPosition:=SR30_CONV_servo_ctrl.Bsetpos , 
	bMoveAbsolute:=SR30_CONV_servo_ctrl.ABSmove_Start , 
	bMoveRelative:=SR30_CONV_servo_ctrl.RELmove_Start , 
	bMoveTorque :=SR30_CONV_servo_ctrl.Torque_mode_Start,
	stManualModeAxis:=SR30_CONV_servo_status , 
	sAxisState=>SR30_CONV_servo_ctrl.Axis_State , 
	bAxis_ready=>SR30_CONV_servo_ctrl.Axis_ready , 
	bAxisInPosition=> SR30_CONV_servo_ctrl.Axis_In_Pos, 
	bAxisError=>SR30_CONV_servo_ctrl.Axis_Error , 
	bAxisEnabled=> SR30_CONV_servo_ctrl.Axis_Enabled, 
	bAxisHomed=> SR30_CONV_servo_ctrl.Axis_reference,
	bTorqueReached=> SR30_CONV_servo_ctrl.Trq_reached, 
	bSetPositionDone=>   ,
	bsafe_to_move=>SR30_CONV_servo_ctrl.Safe_To_Move ,
	bABS_Pos_done=> SR30_CONV_servo_ctrl.pos_done , 
	bHaltDone=> , 
	bSTOPDone=> , 
	bHomeDone=> , 
	bDone=> );	
	
IF OP30_ManualSelected AND MANUAL_SELECTED THEN
	SR30_Vert_servo_status.targetVelocity:=50;
	SR30_Hori_servo_status.targetVelocity:=50;
	//SR30_CONV_servo_status.targetVelocity:=100;
	OP30_GIUDE_GRP_Manual_Axis.targetVelocity:=50;
	OP30_Gripper_LH_Gripper_ctrl.Velocity       :=  500;
	OP30_Gripper_RH_Gripper_ctrl.Velocity       :=  500;
	OP30_Gripper_LH_Gripper_ctrl.ABSmove_Start  :=  LH_Gripper_bMove;
	OP30_Gripper_RH_Gripper_ctrl.ABSmove_Start  :=  RH_Gripper_bMove;	
END_IF

//LH Rejection Cylinder
//move ZERO to STATUS
//CR30_LH_Rej_Cyl_Status:=0;

//Reset Auto Cmd IN Manual Mode & Homing
IF (OP30_Auto OR OP30_HomeRunning) THEN
	CR30_LH_Rej_Cyl.AutoCmd1:=FALSE;
	CR30_LH_Rej_Cyl.AutoCmd2:=FALSE;		
END_IF

// Safe Home
IF (TRUE) AND  (TRUE) THEN 
	CR30_LH_Rej_Cyl.SafeHome:= TRUE ;
ELSE 
	CR30_LH_Rej_Cyl.SafeHome:= FALSE ;
END_IF
// Safe Work
IF (TRUE) OR (TRUE) THEN 
	CR30_LH_Rej_Cyl.Safework:= TRUE ;
ELSE 
	CR30_LH_Rej_Cyl.Safework:= FALSE ;
END_IF
	
// Manual PB  Cyl Mapping
IF (OP30_HMI_LH_Rej_Cyl_Home_PB=TRUE) THEN
	CR30_LH_Rej_Cyl.ManualPB1:=TRUE;
ELSE 
	CR30_LH_Rej_Cyl.ManualPB1:=FALSE;
END_IF
	
IF (OP30_HMI_LH_Rej_Cyl_Work_PB=TRUE) THEN
	CR30_LH_Rej_Cyl.ManualPB2:=TRUE;
ELSE 
	CR30_LH_Rej_Cyl.ManualPB2:=FALSE;
END_IF
	
CR30_LH_Rej_Cyl(
	Auto:= OP30_AutoSelected , 
	Manual:= OP30_ManualSelected AND MANUAL_SELECTED, 
	ErrorActive:= , 
	ResetPB:= OP30_HMI_Reset, 
	Sensor1:= I30_LH_REJ_CYL_FWD_I1100_2, 
	Sensor2:= I30_LH_REJ_CYL_REV_I1100_3,
	ManualPB1:= , 
	ManualPB2:= , 
	AutoCmd1:=CR30_LH_Rej_Cyl_hme , 
	AutoCmd2:=CR30_LH_Rej_Cyl_wrk , 
	OperationEnable:= OperationEnable, 
	SafeHome:= 1, 
	SafeWork:= 1, 
	HomingCmd1:= , 
	Pulse_1Sec:= Pulse_Block.Q1Hz , 
	BlinkingBit:= , 
	TimeOut1:= 5, 
	TimeOut2:= 5, 
	TimeOut3:= 5, 
	Solenoid1=> O30_LH_REJ_CYL_FWD_Q1150_5 , 
	Solenoid2=>  O30_LH_REJ_CYL_REV_Q1150_4 ,
	AlarmSensor1=> , 
	AlarmSensor2=> , 
	AlarmSolenoid1=> , 
	AlarmSolenoid2=> , 
	AllSignal=> , 
	AlarmPresent=> , 
	Position1=> , 
	Position2=> , 
	HomeSensorBlink=> , 
	WorkSensorBlink=> , 
	Status:=CR30_LH_Rej_Cyl_status );


//RH Rejection Cylinder
//move ZERO to STATUS
//CR30_RH_Rej_Cyl_Status:=0;

//Reset Auto Cmd IN Manual Mode & Homing
IF (OP30_Auto OR OP30_HomeRunning) THEN
	CR30_RH_Rej_Cyl.AutoCmd1:=FALSE;
	CR30_RH_Rej_Cyl.AutoCmd2:=FALSE;		
END_IF

// Safe Home
IF (TRUE) AND  (TRUE) THEN 
	CR30_RH_Rej_Cyl.SafeHome:= TRUE ;
ELSE 
	CR30_RH_Rej_Cyl.SafeHome:= FALSE ;
END_IF
// Safe Work
IF (TRUE) OR (TRUE) THEN 
	CR30_RH_Rej_Cyl.Safework:= TRUE ;
ELSE 
	CR30_RH_Rej_Cyl.Safework:= FALSE ;
END_IF
	
// Manual PB  Cyl Mapping
IF (OP30_HMI_RH_Rej_Cyl_Home_PB=TRUE) THEN
	CR30_RH_Rej_Cyl.ManualPB1:=TRUE;
	CR30_RH_Rej_Cyl.ManualPB2:=FALSE;
ELSE 
	CR30_RH_Rej_Cyl.ManualPB1:=FALSE;
END_IF
	
IF (OP30_HMI_RH_Rej_Cyl_Work_PB=TRUE) THEN
	CR30_RH_Rej_Cyl.ManualPB2:=TRUE;
	CR30_RH_Rej_Cyl.ManualPB1:=FALSE;
ELSE 
	CR30_RH_Rej_Cyl.ManualPB2:=FALSE;
END_IF
	
CR30_RH_Rej_Cyl(
	Auto:= OP30_AutoSelected ,  
	Manual:= OP30_ManualSelected AND MANUAL_SELECTED, 
	ErrorActive:= , 
	ResetPB:= OP30_HMI_Reset,                    
	Sensor1:= I30_RH_REJ_CYL_FWD_I1100_4, 
	Sensor2:=  I30_RH_REJ_CYL_REV_I1100_5, 
	ManualPB1:= , 
	ManualPB2:= , 
	AutoCmd1:= CR30_RH_Rej_Cyl_hme, 
	AutoCmd2:= CR30_RH_Rej_Cyl_wrk, 
	OperationEnable:= OperationEnable, 
	SafeHome:= 1, 
	SafeWork:= 1, 
	HomingCmd1:= , 
	Pulse_1Sec:= Pulse_Block.Q1Hz , 
	BlinkingBit:= , 
	TimeOut1:= 5, 
	TimeOut2:= 5, 
	TimeOut3:= 5, 
	Solenoid1=> O30_RH_REJ_CYL_FWD_Q1150_7 , 
	Solenoid2=> O30_RH_REJ_CYL_REV_Q1150_6 , 
	AlarmSensor1=> , 
	AlarmSensor2=> , 
	AlarmSolenoid1=>, 
	AlarmSolenoid2=> , 
	AllSignal=> , 
	AlarmPresent=> , 
	Position1=> , 
	Position2=> , 
	HomeSensorBlink=> , 
	WorkSensorBlink=> , 
	Status:=CR30_RH_Rej_Cyl_status );		
	
OP30_Gripper_LH(
	iHW:= HwIn1 , 
	o_b_enable=> OP30_Gripper_LH_Gripper_ctrl.Axis_Enabled ,
	i_b_moveToPosition:=OP30_Gripper_LH_Gripper_ctrl.ABSmove_Start , 
	i_b_moveRelativ:= , 
	i_b_reference:=OP30_Gripper_LH_Gripper_ctrl.Reference_Start , 
	i_b_ackError:=OP30_HMI_Reset OR Servo_Reset , 
	i_u_targetPos:=OP30_Gripper_LH_Gripper_ctrl.Position , 
	i_u_targetVelocity:=OP30_Gripper_LH_Gripper_ctrl.Velocity , 
	i_u_targetCurrent:= OP30_Gripper_Current , 
	i_u_targetAcceleration:= OP30_Gripper_Acceleration , 
	i_u_targetJerk:= OP30_Gripper_Jerk , 
	i_b_ManualMode:=temp30 , 
	stManualModeAxis:=OP30_Gripper_LH_Manual_Axis , 
	Status=>OP30_Gripper_LH_Gripper_ctrl.Axis_State , 
	o_b_referenced=>OP30_Gripper_LH_Gripper_ctrl.Axis_reference , 
	o_b_reachedPos=> OP30_Gripper_LH_Gripper_ctrl.pos_done , 
	o_u_actualPosition=> OP30_Gripper_LH_Gripper_ctrl.Actual_Position , 
	o_b_error=> OP30_Gripper_LH_Gripper_ctrl.Axis_Error, 
	oHW=> HwOut1 );	
	
OP30_Gripper_RH(
	iHW:= HwIn2 , 
	o_b_enable => OP30_Gripper_RH_Gripper_ctrl.Axis_Enabled,
	i_b_moveToPosition:=OP30_Gripper_RH_Gripper_ctrl.ABSmove_Start , 
	i_b_moveRelativ:= , 
	i_b_reference:=OP30_Gripper_RH_Gripper_ctrl.Reference_Start , 
	i_b_ackError:=OP30_HMI_Reset OR Servo_Reset, 
	i_u_targetPos:=OP30_Gripper_RH_Gripper_ctrl.Position , 
	i_u_targetVelocity:=OP30_Gripper_RH_Gripper_ctrl.Velocity , 
	i_u_targetCurrent:= OP30_Gripper_Current , 
	i_u_targetAcceleration:= OP30_Gripper_Acceleration , 
	i_u_targetJerk:= OP30_Gripper_Jerk , 
	i_b_ManualMode:= temp30, 
	stManualModeAxis:=OP30_Gripper_RH_Manual_Axis , 
	Status=>OP30_Gripper_RH_Gripper_ctrl.Axis_State , 
	o_b_referenced=>OP30_Gripper_RH_Gripper_ctrl.Axis_reference , 
	o_b_reachedPos=> OP30_Gripper_RH_Gripper_ctrl.pos_done , 
	o_u_actualPosition=> OP30_Gripper_RH_Gripper_ctrl.Actual_Position , 
	o_b_error=> OP30_Gripper_RH_Gripper_ctrl.Axis_Error, 
	oHW=> HwOut2 );	

OP30_Gripper_LH_Gripper_ctrl.Velocity       :=  500;
OP30_Gripper_RH_Gripper_ctrl.Velocity       :=  500;	
OP30_Gripper_Current        :=  2;
OP30_Gripper_Acceleration   :=  2500;	
OP30_Gripper_Jerk           :=  50000;

CASE Grip_Test OF
	
	1:  OP30_Gripper_LH_Open:=1;
	   	OP30_Gripper_RH_Open:=1;
	    Grip_Test:=2;	
	   
	2: IF Test.Q THEN
		OP30_Gripper_LH_Close:=1;
		OP30_Gripper_RH_Close:=1;
		Grip_Test:=1;
	   END_IF

END_CASE

Test(IN:= (OP30_Gripper_RH_State AND OP30_Gripper_LH_State), PT:=T#500MS);	

IF Main.EMG_Raise.Q THEN
   Gripper_Ref_Timer.IN:=TRUE;
END_IF
   Gripper_Ref_Timer.PT:=T#5S;
IF Gripper_Ref_Timer.Q THEN
	Gripper_Ref_Timer.IN:=FALSE;
    OP30_Gripper_LH_Gripper_ctrl.Reference_Start:=TRUE;
    OP30_Gripper_RH_Gripper_ctrl.Reference_Start:=TRUE;
END_IF
 
IF OP30_Gripper_LH_Gripper_ctrl.Axis_reference AND OP30_Gripper_LH_Open THEN
	OP30_Gripper_LH_Gripper_ctrl.Position:=OP30_Gripper_Wrk_POS;
	OP30_Gripper_LH_Gripper_ctrl.ABSmove_Start:=TRUE;
	IF OP30_Gripper_LH_Gripper_ctrl.pos_done AND In_range(OP30_Gripper_LH_Gripper_ctrl.Actual_Position,OP30_Gripper_Wrk_POS,1) THEN
		OP30_Gripper_LH_Open:=FALSE;
		OP30_Gripper_LH_Gripper_ctrl.ABSmove_Start:=0;	
		OP30_Gripper_LH_State:=1;
	END_IF
END_IF

IF OP30_Gripper_LH_Gripper_ctrl.Axis_reference AND OP30_Gripper_LH_Close THEN
	OP30_Gripper_LH_Gripper_ctrl.Position:=0;
	OP30_Gripper_LH_Gripper_ctrl.ABSmove_Start:=TRUE;
	IF OP30_Gripper_LH_Gripper_ctrl.pos_done AND In_range(OP30_Gripper_LH_Gripper_ctrl.Actual_Position,0.1,1) THEN
		OP30_Gripper_LH_Close:=FALSE;
		OP30_Gripper_LH_Gripper_ctrl.ABSmove_Start:=0;
		OP30_Gripper_LH_State:=0;
	END_IF
END_IF

